(* CODESYS project PLC_241_14_11_2020.project
   Title: PLC_241
   Version: 0.0.0.0
   Author: anvar

Project tree, tasks and I/O mapping:
  PLC_241 : TM241CE40T/U, Schneider Electric, order no. TM241CE40T/U, version 4.0.6.18
    application Application
      task MAST (cyclic, interval 20 ms, priority 15, watchdog 100 ms x 1) calls BIND, prgLoad, prgLoad_K, prgAdd_weight, CONVERT_REAL_TO_INT, prgDOSING_BIG_WEIGHT, Recept, MotoHours, vsState
      global variables GVL
      global variables IN_OUT
      global variables Mechanizm
      program BIND [ST]
      data type Real_word
      FB/
        SH/
          function block Z [LD]
        Flap/
          function block KP [LD]
        Noria/
          function block N [LD]
        SKTR/
          function block T [LD]
          function block Shnek [LD]
          function block Dozator [LD]
        ASP/
          function block AC [LD]
          function block shluz [LD]
        vibr/
          function block VB [LD]
        scalperator/
          function block SCLP [LD]
      POU/
        program prgLoad [LD]
        program prgLoad_K [LD]
        program prgAdd_weight [LD]
        program prgDOSING_BIG_WEIGHT [LD]
        program MotoHours [ST]
      global variables ErrList
      global variables Pozition_flap
      program Recept [ST]
      program CONVERT_REAL_TO_INT [ST]
      global variables PersistentVars
      program vsState [ST]
      function funStepMH [ST]
    DI : Digital Inputs, Schneider Electric, version 4.0.6.18
        input  idwDI_IDW0 : DWORD  // IDW0
        input  Application.x0_0 : BOOL  // IDW0.I0
        input  Application.x0_1 : BOOL  // IDW0.I1
        input  Application.x0_2 : BOOL  // IDW0.I2
        input  Application.x0_3 : BOOL  // IDW0.I3
        input  Application.x0_4 : BOOL  // IDW0.I4
        input  Application.x0_5 : BOOL  // IDW0.I5
        input  Application.x0_6 : BOOL  // IDW0.I6
        input  Application.x0_7 : BOOL  // IDW0.I7
        input  Application.x0_8 : BOOL  // IDW0.I8
        input  Application.x0_9 : BOOL  // IDW0.I9
        input  Application.x0_10 : BOOL  // IDW0.I10
        input  Application.x0_11 : BOOL  // IDW0.I11
        input  Application.x0_12 : BOOL  // IDW0.I12
        input  Application.x0_13 : BOOL  // IDW0.I13
        input  Application.x0_14 : BOOL  // IDW0.I14
        input  Application.x0_15 : BOOL  // IDW0.I15
        input  Application.x0_16 : BOOL  // IDW0.I16
        input  Application.x0_17 : BOOL  // IDW0.I17
        input  Application.x0_18 : BOOL  // IDW0.I18
        input  Application.x0_19 : BOOL  // IDW0.I19
        input  Application.x0_20 : BOOL  // IDW0.I20
        input  Application.x0_21 : BOOL  // IDW0.I21
        input  Application.x0_22 : BOOL  // IDW0.I22
        input  Application.x0_23 : BOOL  // IDW0.I23
        input  ibDI_IB1 : BYTE  // IB1
    DQ : Digital Outputs, Schneider Electric, version 4.0.6.18
        output Application.y0_0 : BOOL  // QW0.Q0
        output Application.y0_1 : BOOL  // QW0.Q1
        output Application.y0_2 : BOOL  // QW0.Q2
        output Application.y0_3 : BOOL  // QW0.Q3
        output Application.y0_4 : BOOL  // QW0.Q4
        output Application.y0_5 : BOOL  // QW0.Q5
        output Application.y0_6 : BOOL  // QW0.Q6
        output Application.y0_7 : BOOL  // QW0.Q7
        output Application.y0_8 : BOOL  // QW0.Q8
        output Application.y0_9 : BOOL  // QW0.Q9
        output Application.y0_10 : BOOL  // QW0.Q10
        output Application.y0_11 : BOOL  // QW0.Q11
        output Application.y0_12 : BOOL  // QW0.Q12
        output Application.y0_13 : BOOL  // QW0.Q13
        output Application.y0_14 : BOOL  // QW0.Q14
        output Application.y0_15 : BOOL  // QW0.Q15
        output qbDQ_QB1 : BYTE  // QB1
        unmapped channels: QW0
    Counters : Counters, Schneider Electric, version 4.0.6.18
    Pulse_Generators : Pulse Generators, Schneider Electric, version 4.0.6.18
    Cartridge_1 : Cartridge, Schneider Electric, version 4.0.6.18
    Cartridge_2 : Cartridge, Schneider Electric, version 4.0.6.18
    IO_Bus : IO bus - TM3, Schneider Electric, version 4.0.6.18
      IN_1 : TM3DI32K, Schneider Electric, order no. TM3DI32K, version 1.0.1.3
          input  idwIN_1_ID0 : DWORD  // ID0
          input  Application.x1_0 : BOOL  // ID0.I0
          input  Application.x1_1 : BOOL  // ID0.I1
          input  Application.x1_2 : BOOL  // ID0.I2
          input  Application.x1_3 : BOOL  // ID0.I3
          input  Application.x1_4 : BOOL  // ID0.I4
          input  Application.x1_5 : BOOL  // ID0.I5
          input  Application.x1_6 : BOOL  // ID0.I6
          input  Application.x1_7 : BOOL  // ID0.I7
          input  Application.x1_8 : BOOL  // ID0.I8
          input  Application.x1_9 : BOOL  // ID0.I9
          input  Application.x1_10 : BOOL  // ID0.I10
          input  Application.x1_11 : BOOL  // ID0.I11
          input  Application.x1_12 : BOOL  // ID0.I12
          input  Application.x1_13 : BOOL  // ID0.I13
          input  Application.x1_14 : BOOL  // ID0.I14
          input  Application.x1_15 : BOOL  // ID0.I15
          input  Application.x1_16 : BOOL  // ID0.I16
          input  Application.x1_17 : BOOL  // ID0.I17
          input  Application.x1_18 : BOOL  // ID0.I18
          input  Application.x1_19 : BOOL  // ID0.I19
          input  Application.x1_20 : BOOL  // ID0.I20
          input  Application.x1_21 : BOOL  // ID0.I21
          input  Application.x1_22 : BOOL  // ID0.I22
          input  Application.x1_23 : BOOL  // ID0.I23
          input  Application.x1_24 : BOOL  // ID0.I24
          input  Application.x1_25 : BOOL  // ID0.I25
          input  Application.x1_26 : BOOL  // ID0.I26
          input  Application.x1_27 : BOOL  // ID0.I27
          input  Application.x1_28 : BOOL  // ID0.I28
          input  Application.x1_29 : BOOL  // ID0.I29
          input  Application.x1_30 : BOOL  // ID0.I30
          input  Application.x1_31 : BOOL  // ID0.I31
      IN_2 : TM3DI32K, Schneider Electric, order no. TM3DI32K, version 1.0.1.3
          input  idwIN_2_ID0 : DWORD  // ID0
          input  Application.x2_0 : BOOL  // ID0.I0
          input  Application.x2_1 : BOOL  // ID0.I1
          input  Application.x2_2 : BOOL  // ID0.I2
          input  Application.x2_3 : BOOL  // ID0.I3
          input  Application.x2_4 : BOOL  // ID0.I4
          input  Application.x2_5 : BOOL  // ID0.I5
          input  Application.x2_6 : BOOL  // ID0.I6
          input  Application.x2_7 : BOOL  // ID0.I7
          input  Application.x2_8 : BOOL  // ID0.I8
          input  Application.x2_9 : BOOL  // ID0.I9
          input  Application.x2_10 : BOOL  // ID0.I10
          input  Application.x2_11 : BOOL  // ID0.I11
          input  Application.x2_12 : BOOL  // ID0.I12
          input  Application.x2_13 : BOOL  // ID0.I13
          input  Application.x2_14 : BOOL  // ID0.I14
          input  Application.x2_15 : BOOL  // ID0.I15
          input  Application.x2_16 : BOOL  // ID0.I16
          input  Application.x2_17 : BOOL  // ID0.I17
          input  Application.x2_18 : BOOL  // ID0.I18
          input  Application.x2_19 : BOOL  // ID0.I19
          input  Application.x2_20 : BOOL  // ID0.I20
          input  Application.x2_21 : BOOL  // ID0.I21
          input  Application.x2_22 : BOOL  // ID0.I22
          input  Application.x2_23 : BOOL  // ID0.I23
          input  Application.x2_24 : BOOL  // ID0.I24
          input  Application.x2_25 : BOOL  // ID0.I25
          input  Application.x2_26 : BOOL  // ID0.I26
          input  Application.x2_27 : BOOL  // ID0.I27
          input  Application.x2_28 : BOOL  // ID0.I28
          input  Application.x2_29 : BOOL  // ID0.I29
          input  Application.x2_30 : BOOL  // ID0.I30
          input  Application.x2_31 : BOOL  // ID0.I31
      IN_3 : TM3DI32K, Schneider Electric, order no. TM3DI32K, version 1.0.1.3
          input  idwIN_3_ID0 : DWORD  // ID0
          input  Application.x3_0 : BOOL  // ID0.I0
          input  Application.x3_1 : BOOL  // ID0.I1
          input  Application.x3_2 : BOOL  // ID0.I2
          input  Application.x3_3 : BOOL  // ID0.I3
          input  Application.x3_4 : BOOL  // ID0.I4
          input  Application.x3_5 : BOOL  // ID0.I5
          input  Application.x3_6 : BOOL  // ID0.I6
          input  Application.x3_7 : BOOL  // ID0.I7
          input  Application.x3_8 : BOOL  // ID0.I8
          input  Application.x3_9 : BOOL  // ID0.I9
          input  Application.x3_10 : BOOL  // ID0.I10
          input  Application.x3_11 : BOOL  // ID0.I11
          input  Application.x3_12 : BOOL  // ID0.I12
          input  Application.x3_13 : BOOL  // ID0.I13
          input  Application.x3_14 : BOOL  // ID0.I14
          input  Application.x3_15 : BOOL  // ID0.I15
          input  Application.x3_16 : BOOL  // ID0.I16
          input  Application.x3_17 : BOOL  // ID0.I17
          input  Application.x3_18 : BOOL  // ID0.I18
          input  Application.x3_19 : BOOL  // ID0.I19
          input  Application.x3_20 : BOOL  // ID0.I20
          input  Application.x3_21 : BOOL  // ID0.I21
          input  Application.x3_22 : BOOL  // ID0.I22
          input  Application.x3_23 : BOOL  // ID0.I23
          input  Application.x3_24 : BOOL  // ID0.I24
          input  Application.x3_25 : BOOL  // ID0.I25
          input  Application.x3_26 : BOOL  // ID0.I26
          input  Application.x3_27 : BOOL  // ID0.I27
          input  Application.x3_28 : BOOL  // ID0.I28
          input  Application.x3_29 : BOOL  // ID0.I29
          input  Application.x3_30 : BOOL  // ID0.I30
          input  Application.x3_31 : BOOL  // ID0.I31
      IN_4 : TM3DI32K, Schneider Electric, order no. TM3DI32K, version 1.0.1.3
          input  idwIN_4_ID0 : DWORD  // ID0
          input  Application.x4_0 : BOOL  // ID0.I0
          input  Application.x4_1 : BOOL  // ID0.I1
          input  Application.x4_2 : BOOL  // ID0.I2
          input  Application.x4_3 : BOOL  // ID0.I3
          input  Application.x4_4 : BOOL  // ID0.I4
          input  Application.x4_5 : BOOL  // ID0.I5
          input  Application.x4_6 : BOOL  // ID0.I6
          input  Application.x4_7 : BOOL  // ID0.I7
          input  Application.x4_8 : BOOL  // ID0.I8
          input  Application.x4_9 : BOOL  // ID0.I9
          input  Application.x4_10 : BOOL  // ID0.I10
          input  Application.x4_11 : BOOL  // ID0.I11
          input  Application.x4_12 : BOOL  // ID0.I12
          input  Application.x4_13 : BOOL  // ID0.I13
          input  Application.x4_14 : BOOL  // ID0.I14
          input  Application.x4_15 : BOOL  // ID0.I15
          input  Application.x4_16 : BOOL  // ID0.I16
          input  Application.x4_17 : BOOL  // ID0.I17
          input  Application.x4_18 : BOOL  // ID0.I18
          input  Application.x4_19 : BOOL  // ID0.I19
          input  Application.x4_20 : BOOL  // ID0.I20
          input  Application.x4_21 : BOOL  // ID0.I21
          input  Application.x4_22 : BOOL  // ID0.I22
          input  Application.x4_23 : BOOL  // ID0.I23
          input  Application.x4_24 : BOOL  // ID0.I24
          input  Application.x4_25 : BOOL  // ID0.I25
          input  Application.x4_26 : BOOL  // ID0.I26
          input  Application.x4_27 : BOOL  // ID0.I27
          input  Application.x4_28 : BOOL  // ID0.I28
          input  Application.x4_29 : BOOL  // ID0.I29
          input  Application.x4_30 : BOOL  // ID0.I30
          input  Application.x4_31 : BOOL  // ID0.I31
      IN_5 : TM3DI32K, Schneider Electric, order no. TM3DI32K, version 1.0.1.3
          input  idwIN_5_ID0 : DWORD  // ID0
          input  Application.x5_0 : BOOL  // ID0.I0
          input  Application.x5_1 : BOOL  // ID0.I1
          input  Application.x5_2 : BOOL  // ID0.I2
          input  Application.x5_3 : BOOL  // ID0.I3
          input  Application.x5_4 : BOOL  // ID0.I4
          input  Application.x5_5 : BOOL  // ID0.I5
          input  Application.x5_6 : BOOL  // ID0.I6
          input  Application.x5_7 : BOOL  // ID0.I7
          input  Application.x5_8 : BOOL  // ID0.I8
          input  Application.x5_9 : BOOL  // ID0.I9
          input  Application.x5_10 : BOOL  // ID0.I10
          input  Application.x5_11 : BOOL  // ID0.I11
          input  Application.x5_12 : BOOL  // ID0.I12
          input  Application.x5_13 : BOOL  // ID0.I13
          input  Application.x5_14 : BOOL  // ID0.I14
          input  Application.x5_15 : BOOL  // ID0.I15
          input  Application.x5_16 : BOOL  // ID0.I16
          input  Application.x5_17 : BOOL  // ID0.I17
          input  Application.x5_18 : BOOL  // ID0.I18
          input  Application.x5_19 : BOOL  // ID0.I19
          input  Application.x5_20 : BOOL  // ID0.I20
          input  Application.x5_21 : BOOL  // ID0.I21
          input  Application.x5_22 : BOOL  // ID0.I22
          input  Application.x5_23 : BOOL  // ID0.I23
          input  Application.x5_24 : BOOL  // ID0.I24
          input  Application.x5_25 : BOOL  // ID0.I25
          input  Application.x5_26 : BOOL  // ID0.I26
          input  Application.x5_27 : BOOL  // ID0.I27
          input  Application.x5_28 : BOOL  // ID0.I28
          input  Application.x5_29 : BOOL  // ID0.I29
          input  Application.x5_30 : BOOL  // ID0.I30
          input  Application.x5_31 : BOOL  // ID0.I31
      OUT_6 : TM3DQ32TK, Schneider Electric, order no. TM3DQ32TK, version 1.0.1.3
          output Application.y6_0 : BOOL  // QD0.Q0
          output Application.y6_1 : BOOL  // QD0.Q1
          output Application.y6_2 : BOOL  // QD0.Q2
          output Application.y6_3 : BOOL  // QD0.Q3
          output Application.y6_4 : BOOL  // QD0.Q4
          output Application.y6_5 : BOOL  // QD0.Q5
          output Application.y6_6 : BOOL  // QD0.Q6
          output Application.y6_7 : BOOL  // QD0.Q7
          output Application.y6_8 : BOOL  // QD0.Q8
          output Application.y6_9 : BOOL  // QD0.Q9
          output Application.y6_10 : BOOL  // QD0.Q10
          output Application.y6_11 : BOOL  // QD0.Q11
          output Application.y6_12 : BOOL  // QD0.Q12
          output Application.y6_13 : BOOL  // QD0.Q13
          output Application.y6_14 : BOOL  // QD0.Q14
          output Application.y6_15 : BOOL  // QD0.Q15
          output Application.y6_16 : BOOL  // QD0.Q16
          output Application.y6_17 : BOOL  // QD0.Q17
          output Application.y6_18 : BOOL  // QD0.Q18
          output Application.y6_19 : BOOL  // QD0.Q19
          output Application.y6_20 : BOOL  // QD0.Q20
          output Application.y6_21 : BOOL  // QD0.Q21
          output Application.y6_22 : BOOL  // QD0.Q22
          output Application.y6_23 : BOOL  // QD0.Q23
          output Application.y6_24 : BOOL  // QD0.Q24
          output Application.y6_25 : BOOL  // QD0.Q25
          output Application.y6_26 : BOOL  // QD0.Q26
          output Application.y6_27 : BOOL  // QD0.Q27
          output Application.y6_28 : BOOL  // QD0.Q28
          output Application.y6_29 : BOOL  // QD0.Q29
          output Application.y6_30 : BOOL  // QD0.Q30
          output Application.y6_31 : BOOL  // QD0.Q31
          unmapped channels: QD0
      OUT_7 : TM3DQ32TK, Schneider Electric, order no. TM3DQ32TK, version 1.0.1.3
          output Application.y7_0 : BOOL  // QD0.Q0
          output Application.y7_1 : BOOL  // QD0.Q1
          output Application.y7_2 : BOOL  // QD0.Q2
          output Application.y7_3 : BOOL  // QD0.Q3
          output Application.y7_4 : BOOL  // QD0.Q4
          output Application.y7_5 : BOOL  // QD0.Q5
          output Application.y7_6 : BOOL  // QD0.Q6
          output Application.y7_7 : BOOL  // QD0.Q7
          output Application.y7_8 : BOOL  // QD0.Q8
          output Application.y7_9 : BOOL  // QD0.Q9
          output Application.y7_10 : BOOL  // QD0.Q10
          output Application.y7_11 : BOOL  // QD0.Q11
          output Application.y7_12 : BOOL  // QD0.Q12
          output Application.y7_13 : BOOL  // QD0.Q13
          output Application.y7_14 : BOOL  // QD0.Q14
          output Application.y7_15 : BOOL  // QD0.Q15
          output Application.y7_16 : BOOL  // QD0.Q16
          output Application.y7_17 : BOOL  // QD0.Q17
          output Application.y7_18 : BOOL  // QD0.Q18
          output Application.y7_19 : BOOL  // QD0.Q19
          output Application.y7_20 : BOOL  // QD0.Q20
          output Application.y7_21 : BOOL  // QD0.Q21
          output Application.y7_22 : BOOL  // QD0.Q22
          output Application.y7_23 : BOOL  // QD0.Q23
          output Application.y7_24 : BOOL  // QD0.Q24
          output Application.y7_25 : BOOL  // QD0.Q25
          output Application.y7_26 : BOOL  // QD0.Q26
          output Application.y7_27 : BOOL  // QD0.Q27
          output Application.y7_28 : BOOL  // QD0.Q28
          output Application.y7_29 : BOOL  // QD0.Q29
          output Application.y7_30 : BOOL  // QD0.Q30
          output Application.y7_31 : BOOL  // QD0.Q31
          unmapped channels: QD0
    COM_Bus : COM bus, Schneider Electric, version 4.0.6.18
    Ethernet_1 : Ethernet Network, Schneider Electric, version 4.0.6.18
        settings: IPAddress = [192, 168, 3, 241]; SubnetMask = [255, 255, 255, 0]; WebServer = TRUE; FTP Server = TRUE; SoMachine Protocol = TRUE; Modbus Server = TRUE; NetManage Protocol = TRUE; SNMP protocol = TRUE; Enable Routing = FALSE; WebVisu protocol = TRUE; DHCP Server Active = TRUE
      Ethernet_Manager : Industrial Ethernet Manager, Schneider Electric, version 1.0.12.21
          settings: BinaryFileSize = 396; Dhcps Host 0.Client Mac Address = [16#0, 16#0, 16#0, 16#0, 16#0]; Dhcps Host 0.Client Device Name = 'DEVICE_1'; Dhcps Host 0.Client IP Address = [192, 168, 3, 221]; Dhcps Host 0.Network Mask = [255, 255, 255, 0]; Dhcps Host 0.Default Gateway = [192, 168, 3, 241]; Dhcps Host 1.Client Mac Address = [16#0, 16#0, 16#0, 16#0, 16#0]; Dhcps Host 2.Client Mac Address = [16#0, 16#0, 16#0, 16#0, 16#0]; Dhcps Host 3.Client Mac Address = [16#0, 16#0, 16#0, 16#0, 16#0]; Dhcps Host 4.Client Mac Address = [16#0, 16#0, 16#0, 16#0, 16#0]; Dhcps Host 5.Client Mac Address = [16#0, 16#0, 16#0, 16#0, 16#0]; Dhcps Host 6.Client Mac Address = [16#0, 16#0, 16#0, 16#0, 16#0]; Dhcps Host 7.Client Mac Address = [16#0, 16#0, 16#0, 16#0, 16#0]; Dhcps Host 8.Client Mac Address = [16#0, 16#0, 16#0, 16#0, 16#0]; Dhcps Host 9.Client Mac Address = [16#0, 16#0, 16#0, 16#0, 16#0]; Dhcps Host 10.Client Mac Address = [16#0, 16#0, 16#0, 16#0, 16#0]; Dhcps Host 11.Client Mac Address = [16#0, 16#0, 16#0, 16#0, 16#0]; Dhcps Host 12.Client Mac Address = [16#0, 16#0, 16#0, 16#0, 16#0]; Dhcps Host 13.Client Mac Address = [16#0, 16#0, 16#0, 16#0, 16#0]; Dhcps Host 14.Client Mac Address = [16#0, 16#0, 16#0, 16#0, 16#0]; Dhcps Host 15.Client Mac Address = [16#0, 16#0, 16#0, 16#0, 16#0]; Dhcps Host 16.Client Mac Address = [16#0, 16#0, 16#0, 16#0, 16#0]; Dhcps Host 17.Client Mac Address = [16#0, 16#0, 16#0, 16#0, 16#0]; Dhcps Host 18.Client Mac Address = [16#0, 16#0, 16#0, 16#0, 16#0]; Dhcps Host 19.Client Mac Address = [16#0, 16#0, 16#0, 16#0, 16#0]; Dhcps Host 20.Client Mac Address = [16#0, 16#0, 16#0, 16#0, 16#0]; Dhcps Host 21.Client Mac Address = [16#0, 16#0, 16#0, 16#0, 16#0]; Dhcps Host 22.Client Mac Address = [16#0, 16#0, 16#0, 16#0, 16#0]; Dhcps Host 23.Client Mac Address = [16#0, 16#0, 16#0, 16#0, 16#0]; Dhcps Host 24.Client Mac Address = [16#0, 16#0, 16#0, 16#0, 16#0]; Dhcps Host 25.Client Mac Address = [16#0, 16#0, 16#0, 16#0, 16#0]; Dhcps Host 26.Client Mac Address = [16#0, 16#0, 16#0, 16#0, 16#0]; Dhcps Host 27.Client Mac Address = [16#0, 16#0, 16#0, 16#0, 16#0]; Dhcps Host 28.Client Mac Address = [16#0, 16#0, 16#0, 16#0, 16#0]; Dhcps Host 29.Client Mac Address = [16#0, 16#0, 16#0, 16#0, 16#0]; Dhcps Host 30.Client Mac Address = [16#0, 16#0, 16#0, 16#0, 16#0]; Dhcps Host 31.Client Mac Address = [16#0, 16#0, 16#0, 16#0, 16#0]; Dhcps Host 32.Client Mac Address = [16#0, 16#0, 16#0, 16#0, 16#0]; Dhcps Host 33.Client Mac Address = [16#0, 16#0, 16#0, 16#0, 16#0]; Dhcps Host 34.Client Mac Address = [16#0, 16#0, 16#0, 16#0, 16#0];
            Dhcps Host 35.Client Mac Address = [16#0, 16#0, 16#0, 16#0, 16#0]; Dhcps Host 36.Client Mac Address = [16#0, 16#0, 16#0, 16#0, 16#0]; Dhcps Host 37.Client Mac Address = [16#0, 16#0, 16#0, 16#0, 16#0]; Dhcps Host 38.Client Mac Address = [16#0, 16#0, 16#0, 16#0, 16#0]; Dhcps Host 39.Client Mac Address = [16#0, 16#0, 16#0, 16#0, 16#0]; Dhcps Host 40.Client Mac Address = [16#0, 16#0, 16#0, 16#0, 16#0]; Dhcps Host 41.Client Mac Address = [16#0, 16#0, 16#0, 16#0, 16#0]; Dhcps Host 42.Client Mac Address = [16#0, 16#0, 16#0, 16#0, 16#0]; Dhcps Host 43.Client Mac Address = [16#0, 16#0, 16#0, 16#0, 16#0]; Dhcps Host 44.Client Mac Address = [16#0, 16#0, 16#0, 16#0, 16#0]; Dhcps Host 45.Client Mac Address = [16#0, 16#0, 16#0, 16#0, 16#0]; Dhcps Host 46.Client Mac Address = [16#0, 16#0, 16#0, 16#0, 16#0]; Dhcps Host 47.Client Mac Address = [16#0, 16#0, 16#0, 16#0, 16#0]; Dhcps Host 48.Client Mac Address = [16#0, 16#0, 16#0, 16#0, 16#0]; Dhcps Host 49.Client Mac Address = [16#0, 16#0, 16#0, 16#0, 16#0]; Dhcps Host 50.Client Mac Address = [16#0, 16#0, 16#0, 16#0, 16#0]; Dhcps Host 51.Client Mac Address = [16#0, 16#0, 16#0, 16#0, 16#0]; Dhcps Host 52.Client Mac Address = [16#0, 16#0, 16#0, 16#0, 16#0]; Dhcps Host 53.Client Mac Address = [16#0, 16#0, 16#0, 16#0, 16#0]; Dhcps Host 54.Client Mac Address = [16#0, 16#0, 16#0, 16#0, 16#0]; Dhcps Host 55.Client Mac Address = [16#0, 16#0, 16#0, 16#0, 16#0]; Dhcps Host 56.Client Mac Address = [16#0, 16#0, 16#0, 16#0, 16#0]; Dhcps Host 57.Client Mac Address = [16#0, 16#0, 16#0, 16#0, 16#0]; Dhcps Host 58.Client Mac Address = [16#0, 16#0, 16#0, 16#0, 16#0]; Dhcps Host 59.Client Mac Address = [16#0, 16#0, 16#0, 16#0, 16#0]; Dhcps Host 60.Client Mac Address = [16#0, 16#0, 16#0, 16#0, 16#0]; Dhcps Host 61.Client Mac Address = [16#0, 16#0, 16#0, 16#0, 16#0]; Dhcps Host 62.Client Mac Address = [16#0, 16#0, 16#0, 16#0, 16#0]; Dhcps Host 63.Client Mac Address = [16#0, 16#0, 16#0, 16#0, 16#0]; Dhcps Host 64.Client Mac Address = [16#0, 16#0, 16#0, 16#0, 16#0]; Dhcps Host 65.Client Mac Address = [16#0, 16#0, 16#0, 16#0, 16#0]; Dhcps Host 66.Client Mac Address = [16#0, 16#0, 16#0, 16#0, 16#0]; Dhcps Host 67.Client Mac Address = [16#0, 16#0, 16#0, 16#0, 16#0]; Dhcps Host 68.Client Mac Address = [16#0, 16#0, 16#0, 16#0, 16#0]; Dhcps Host 69.Client Mac Address = [16#0, 16#0, 16#0, 16#0, 16#0]; Dhcps Host 70.Client Mac Address = [16#0, 16#0, 16#0, 16#0, 16#0]; Dhcps Host 71.Client Mac Address = [16#0, 16#0, 16#0, 16#0, 16#0]; Dhcps Host 72.Client Mac Address = [16#0, 16#0, 16#0, 16#0, 16#0]; Dhcps Host 73.Client Mac Address = [16#0, 16#0, 16#0, 16#0, 16#0]; Dhcps Host 74.Client Mac Address = [16#0, 16#0, 16#0, 16#0, 16#0];
            Dhcps Host 75.Client Mac Address = [16#0, 16#0, 16#0, 16#0, 16#0]; Dhcps Host 76.Client Mac Address = [16#0, 16#0, 16#0, 16#0, 16#0]; Dhcps Host 77.Client Mac Address = [16#0, 16#0, 16#0, 16#0, 16#0]; Dhcps Host 78.Client Mac Address = [16#0, 16#0, 16#0, 16#0, 16#0]; Dhcps Host 79.Client Mac Address = [16#0, 16#0, 16#0, 16#0, 16#0]; Dhcps Host 80.Client Mac Address = [16#0, 16#0, 16#0, 16#0, 16#0]; Dhcps Host 81.Client Mac Address = [16#0, 16#0, 16#0, 16#0, 16#0]; Dhcps Host 82.Client Mac Address = [16#0, 16#0, 16#0, 16#0, 16#0]; Dhcps Host 83.Client Mac Address = [16#0, 16#0, 16#0, 16#0, 16#0]; Dhcps Host 84.Client Mac Address = [16#0, 16#0, 16#0, 16#0, 16#0]; Dhcps Host 85.Client Mac Address = [16#0, 16#0, 16#0, 16#0, 16#0]; Dhcps Host 86.Client Mac Address = [16#0, 16#0, 16#0, 16#0, 16#0]; Dhcps Host 87.Client Mac Address = [16#0, 16#0, 16#0, 16#0, 16#0]; Dhcps Host 88.Client Mac Address = [16#0, 16#0, 16#0, 16#0, 16#0]; Dhcps Host 89.Client Mac Address = [16#0, 16#0, 16#0, 16#0, 16#0]; Dhcps Host 90.Client Mac Address = [16#0, 16#0, 16#0, 16#0, 16#0]; Dhcps Host 91.Client Mac Address = [16#0, 16#0, 16#0, 16#0, 16#0]; Dhcps Host 92.Client Mac Address = [16#0, 16#0, 16#0, 16#0, 16#0]; Dhcps Host 93.Client Mac Address = [16#0, 16#0, 16#0, 16#0, 16#0]; Dhcps Host 94.Client Mac Address = [16#0, 16#0, 16#0, 16#0, 16#0]; Dhcps Host 95.Client Mac Address = [16#0, 16#0, 16#0, 16#0, 16#0]; Dhcps Host 96.Client Mac Address = [16#0, 16#0, 16#0, 16#0, 16#0]; Dhcps Host 97.Client Mac Address = [16#0, 16#0, 16#0, 16#0, 16#0]; Dhcps Host 98.Client Mac Address = [16#0, 16#0, 16#0, 16#0, 16#0]; Dhcps Host 99.Client Mac Address = [16#0, 16#0, 16#0, 16#0, 16#0]; Dhcps Host 100.Client Mac Address = [16#0, 16#0, 16#0, 16#0, 16#0]; Dhcps Host 101.Client Mac Address = [16#0, 16#0, 16#0, 16#0, 16#0]; Dhcps Host 102.Client Mac Address = [16#0, 16#0, 16#0, 16#0, 16#0]; Dhcps Host 103.Client Mac Address = [16#0, 16#0, 16#0, 16#0, 16#0]; Dhcps Host 104.Client Mac Address = [16#0, 16#0, 16#0, 16#0, 16#0]; Dhcps Host 105.Client Mac Address = [16#0, 16#0, 16#0, 16#0, 16#0]; Dhcps Host 106.Client Mac Address = [16#0, 16#0, 16#0, 16#0, 16#0]; Dhcps Host 107.Client Mac Address = [16#0, 16#0, 16#0, 16#0, 16#0]; Dhcps Host 108.Client Mac Address = [16#0, 16#0, 16#0, 16#0, 16#0]; Dhcps Host 109.Client Mac Address = [16#0, 16#0, 16#0, 16#0, 16#0]; Dhcps Host 110.Client Mac Address = [16#0, 16#0, 16#0, 16#0, 16#0]; Dhcps Host 111.Client Mac Address = [16#0, 16#0, 16#0, 16#0, 16#0]; Dhcps Host 112.Client Mac Address = [16#0, 16#0, 16#0, 16#0, 16#0]; Dhcps Host 113.Client Mac Address = [16#0, 16#0, 16#0, 16#0, 16#0]; Dhcps Host 114.Client Mac Address = [16#0, 16#0, 16#0, 16#0, 16#0];
            Dhcps Host 115.Client Mac Address = [16#0, 16#0, 16#0, 16#0, 16#0]; Dhcps Host 116.Client Mac Address = [16#0, 16#0, 16#0, 16#0, 16#0]; Dhcps Host 117.Client Mac Address = [16#0, 16#0, 16#0, 16#0, 16#0]; Dhcps Host 118.Client Mac Address = [16#0, 16#0, 16#0, 16#0, 16#0]; Dhcps Host 119.Client Mac Address = [16#0, 16#0, 16#0, 16#0, 16#0]; Dhcps Host 120.Client Mac Address = [16#0, 16#0, 16#0, 16#0, 16#0]; Dhcps Host 121.Client Mac Address = [16#0, 16#0, 16#0, 16#0, 16#0]; Dhcps Host 122.Client Mac Address = [16#0, 16#0, 16#0, 16#0, 16#0]; Dhcps Host 123.Client Mac Address = [16#0, 16#0, 16#0, 16#0, 16#0]; Dhcps Host 124.Client Mac Address = [16#0, 16#0, 16#0, 16#0, 16#0]; Dhcps Host 125.Client Mac Address = [16#0, 16#0, 16#0, 16#0, 16#0]; Dhcps Host 126.Client Mac Address = [16#0, 16#0, 16#0, 16#0, 16#0]; Dhcps Host 127.Client Mac Address = [16#0, 16#0, 16#0, 16#0, 16#0]; Dhcps Host 128.Client Mac Address = [16#0, 16#0, 16#0, 16#0, 16#0]; serialized Values = 9e259374-7d59-4259-90d2-1eb457ee1159=0|
          unmapped channels: Global Status, Healthbit 0, Healthbit 1, Healthbit 2, Healthbit 3
        Modbus_TCP_Slave_PLC221 : Generic Modbus TCP Slave, Schneider Electric, version 1.0.2.21
            settings: Unit-ID = 248; IPAddress = [192, 168, 3, 221]; GatewayAddress = [192, 168, 3, 241]; DeviceName = 'DEVICE_1'; PLC221.Channel ID = 0; PLC221.Unit-ID = 255; PLC221.Repetition Rate = 20; PLC221.Function Code = 23; PLC221.Read Offset = 16#0000; PLC221.Read Length = 20; PLC221.Write Offset = 16#0014; PLC221.Write Length = 10
            input  Application.a2x0_0 : BOOL  // PLC221.Bit 0
            input  Application.a2x0_1 : BOOL  // PLC221.Bit 1
            input  Application.a2x0_2 : BOOL  // PLC221.Bit 2
            input  Application.a2x0_3 : BOOL  // PLC221.Bit 3
            input  Application.a2x0_4 : BOOL  // PLC221.Bit 4
            input  Application.a2x0_5 : BOOL  // PLC221.Bit 5
            input  Application.a2x0_6 : BOOL  // PLC221.Bit 6
            input  Application.a2x0_7 : BOOL  // PLC221.Bit 7
            input  Application.a2x0_8 : BOOL  // PLC221.Bit 8
            input  Application.a2x0_9 : BOOL  // PLC221.Bit 9
            input  Application.a2x0_10 : BOOL  // PLC221.Bit 10
            input  Application.a2x0_11 : BOOL  // PLC221.Bit 11
            input  Application.a2x0_12 : BOOL  // PLC221.Bit 12
            input  Application.a2x0_13 : BOOL  // PLC221.Bit 13
            input  Application.a2x0_14 : BOOL  // PLC221.Bit 14
            input  Application.a2x0_15 : BOOL  // PLC221.Bit 15
            input  Application.a2x0_16 : BOOL  // PLC221.Bit 0
            input  Application.a2x0_17 : BOOL  // PLC221.Bit 1
            input  Application.a2x0_18 : BOOL  // PLC221.Bit 2
            input  Application.a2x0_19 : BOOL  // PLC221.Bit 3
            input  Application.a2x0_20 : BOOL  // PLC221.Bit 4
            input  Application.a2x0_21 : BOOL  // PLC221.Bit 5
            input  Application.a2x0_22 : BOOL  // PLC221.Bit 6
            input  Application.a2x0_23 : BOOL  // PLC221.Bit 7
            input  Application.a2x3_0 : BOOL  // PLC221.Bit 0
            input  Application.a2x3_1 : BOOL  // PLC221.Bit 1
            input  Application.a2x3_2 : BOOL  // PLC221.Bit 2
            input  Application.a2x3_3 : BOOL  // PLC221.Bit 3
            input  Application.a2x3_4 : BOOL  // PLC221.Bit 4
            input  Application.a2x3_5 : BOOL  // PLC221.Bit 5
            input  Application.a2x3_6 : BOOL  // PLC221.Bit 6
            input  Application.a2x3_7 : BOOL  // PLC221.Bit 7
            input  Application.a2x3_8 : BOOL  // PLC221.Bit 8
            input  Application.a2x3_9 : BOOL  // PLC221.Bit 9
            input  Application.a2x3_10 : BOOL  // PLC221.Bit 10
            input  Application.a2x3_11 : BOOL  // PLC221.Bit 11
            input  Application.a2x3_12 : BOOL  // PLC221.Bit 12
            input  Application.a2x3_13 : BOOL  // PLC221.Bit 13
            input  Application.a2x3_14 : BOOL  // PLC221.Bit 14
            input  Application.a2x3_15 : BOOL  // PLC221.Bit 15
            input  Application.a2x3_16 : BOOL  // PLC221.Bit 0
            input  Application.a2x3_17 : BOOL  // PLC221.Bit 1
            input  Application.a2x3_18 : BOOL  // PLC221.Bit 2
            input  Application.a2x3_19 : BOOL  // PLC221.Bit 3
            input  Application.a2x3_20 : BOOL  // PLC221.Bit 4
            input  Application.a2x3_21 : BOOL  // PLC221.Bit 5
            input  Application.a2x3_22 : BOOL  // PLC221.Bit 6
            input  Application.a2x3_23 : BOOL  // PLC221.Bit 7
            input  Application.a2x3_24 : BOOL  // PLC221.Bit 8
            input  Application.a2x3_25 : BOOL  // PLC221.Bit 9
            input  Application.a2x3_26 : BOOL  // PLC221.Bit 10
            input  Application.a2x3_27 : BOOL  // PLC221.Bit 11
            input  Application.a2x3_28 : BOOL  // PLC221.Bit 12
            input  Application.a2x3_29 : BOOL  // PLC221.Bit 13
            input  Application.a2x3_30 : BOOL  // PLC221.Bit 14
            input  Application.a2x3_31 : BOOL  // PLC221.Bit 15
            input  Application.a2x4_0 : BOOL  // PLC221.Bit 0
            input  Application.a2x4_1 : BOOL  // PLC221.Bit 1
            input  Application.a2x4_2 : BOOL  // PLC221.Bit 2
            input  Application.a2x4_3 : BOOL  // PLC221.Bit 3
            input  Application.a2x4_4 : BOOL  // PLC221.Bit 4
            input  Application.a2x4_5 : BOOL  // PLC221.Bit 5
            input  Application.a2x4_6 : BOOL  // PLC221.Bit 6
            input  Application.a2x4_7 : BOOL  // PLC221.Bit 7
            input  Application.a2x4_8 : BOOL  // PLC221.Bit 8
            input  Application.a2x4_9 : BOOL  // PLC221.Bit 9
            input  Application.a2x4_10 : BOOL  // PLC221.Bit 10
            input  Application.a2x4_11 : BOOL  // PLC221.Bit 11
            input  Application.a2x4_12 : BOOL  // PLC221.Bit 12
            input  Application.a2x4_13 : BOOL  // PLC221.Bit 13
            input  Application.a2x4_14 : BOOL  // PLC221.Bit 14
            input  Application.a2x4_15 : BOOL  // PLC221.Bit 15
            input  Application.a2x4_16 : BOOL  // PLC221.Bit 0
            input  Application.a2x4_17 : BOOL  // PLC221.Bit 1
            input  Application.a2x4_18 : BOOL  // PLC221.Bit 2
            input  Application.a2x4_19 : BOOL  // PLC221.Bit 3
            input  Application.a2x4_20 : BOOL  // PLC221.Bit 4
            input  Application.a2x4_21 : BOOL  // PLC221.Bit 5
            input  Application.a2x4_22 : BOOL  // PLC221.Bit 6
            input  Application.a2x4_23 : BOOL  // PLC221.Bit 7
            input  Application.a2x4_24 : BOOL  // PLC221.Bit 8
            input  Application.a2x4_25 : BOOL  // PLC221.Bit 9
            input  Application.a2x4_26 : BOOL  // PLC221.Bit 10
            input  Application.a2x4_27 : BOOL  // PLC221.Bit 11
            input  Application.a2x4_28 : BOOL  // PLC221.Bit 12
            input  Application.a2x4_29 : BOOL  // PLC221.Bit 13
            input  Application.a2x4_30 : BOOL  // PLC221.Bit 14
            input  Application.a2x4_31 : BOOL  // PLC221.Bit 15
            input  Application.a2x5_0 : BOOL  // PLC221.Bit 0
            input  Application.a2x5_1 : BOOL  // PLC221.Bit 1
            input  Application.a2x5_2 : BOOL  // PLC221.Bit 2
            input  Application.a2x5_3 : BOOL  // PLC221.Bit 3
            input  Application.a2x5_4 : BOOL  // PLC221.Bit 4
            input  Application.a2x5_5 : BOOL  // PLC221.Bit 5
            input  Application.a2x5_6 : BOOL  // PLC221.Bit 6
            input  Application.a2x5_7 : BOOL  // PLC221.Bit 7
            input  Application.a2x5_8 : BOOL  // PLC221.Bit 8
            input  Application.a2x5_9 : BOOL  // PLC221.Bit 9
            input  Application.a2x5_10 : BOOL  // PLC221.Bit 10
            input  Application.a2x5_11 : BOOL  // PLC221.Bit 11
            input  Application.a2x5_12 : BOOL  // PLC221.Bit 12
            input  Application.a2x5_13 : BOOL  // PLC221.Bit 13
            input  Application.a2x5_14 : BOOL  // PLC221.Bit 14
            input  Application.a2x5_15 : BOOL  // PLC221.Bit 15
            input  Application.a2x5_16 : BOOL  // PLC221.Bit 0
            input  Application.a2x5_17 : BOOL  // PLC221.Bit 1
            input  Application.a2x5_18 : BOOL  // PLC221.Bit 2
            input  Application.a2x5_19 : BOOL  // PLC221.Bit 3
            input  Application.a2x5_20 : BOOL  // PLC221.Bit 4
            input  Application.a2x5_21 : BOOL  // PLC221.Bit 5
            input  Application.a2x5_22 : BOOL  // PLC221.Bit 6
            input  Application.a2x5_23 : BOOL  // PLC221.Bit 7
            input  Application.a2x5_24 : BOOL  // PLC221.Bit 8
            input  Application.a2x5_25 : BOOL  // PLC221.Bit 9
            input  Application.a2x5_26 : BOOL  // PLC221.Bit 10
            input  Application.a2x5_27 : BOOL  // PLC221.Bit 11
            input  Application.a2x5_28 : BOOL  // PLC221.Bit 12
            input  Application.a2x5_29 : BOOL  // PLC221.Bit 13
            input  Application.a2x5_30 : BOOL  // PLC221.Bit 14
            input  Application.a2x5_31 : BOOL  // PLC221.Bit 15
            input  Application.IW1_0 : WORD  // PLC221
            input  Application.IW1_1 : WORD  // PLC221
            input  Application.IW1_2 : WORD  // PLC221
            input  Application.IW1_3 : WORD  // PLC221
            input  Application.IW2_0 : WORD  // PLC221
            unmapped channels: PLC221, PLC221, PLC221, PLC221, PLC221, PLC221, PLC221, PLC221, PLC221, PLC221, PLC221, PLC221, PLC221, PLC221, PLC221, PLC221, PLC221, PLC221, PLC221, PLC221, PLC221, PLC221, PLC221, PLC221, PLC221
    Serial_Line_1 : Serial line, Schneider Electric, version 4.0.6.18
      Pch : Modbus IOScanner, Schneider Electric, version 3.5.3.8
        PCH_BIG_11_16 : Generic Modbus Slave, Schneider Electric, version 3.5.3.9
            settings: SlaveAddress = 2; ResponseTimeout = 1000; Channel 1.Function Code = 6; Channel 1.Read Offset = 0; Channel 1.Read Length = 0; Channel 1.Write Offset = 16#FA01; Channel 1.Write Length = 1; Channel 1.Cycle Time = 20; Channel 2.Function Code = 3; Channel 2.Read Offset = 16#FD00; Channel 2.Read Length = 1; Channel 2.Write Offset = 0; Channel 2.Write Length = 0; Channel 2.Cycle Time = 100; Channel 3.Function Code = 3; Channel 3.Read Offset = 16#FE03; Channel 3.Read Length = 1; Channel 3.Write Offset = 0; Channel 3.Write Length = 0; Channel 3.Cycle Time = 100
            output WrFreq_pch_big_11_16 : ARRAY[0..0] OF WORD  // Channel 1
            input  ReadFreq_pch_big_11_16 : ARRAY[0..0] OF WORD  // Channel 2
            input  ReadCurr_pch_big_11_16 : ARRAY[0..0] OF WORD  // Channel 3
        PCH_BIG_17_18 : Generic Modbus Slave, Schneider Electric, version 3.5.3.9
            settings: SlaveAddress = 3; ResponseTimeout = 1000; Channel 1.Function Code = 6; Channel 1.Read Offset = 0; Channel 1.Read Length = 0; Channel 1.Write Offset = 16#FA01; Channel 1.Write Length = 1; Channel 1.Cycle Time = 20; Channel 2.Function Code = 3; Channel 2.Read Offset = 16#FD00; Channel 2.Read Length = 1; Channel 2.Write Offset = 0; Channel 2.Write Length = 0; Channel 2.Cycle Time = 100; Channel 3.Function Code = 3; Channel 3.Read Offset = 16#FE03; Channel 3.Read Length = 1; Channel 3.Write Offset = 0; Channel 3.Write Length = 0; Channel 3.Cycle Time = 100
            output WrFreq_pch_big_17_18 : ARRAY[0..0] OF WORD  // Channel 1
            input  ReadFreq_pch_big_17_18 : ARRAY[0..0] OF WORD  // Channel 2
            input  ReadCurr_pch_big_17_18 : ARRAY[0..0] OF WORD  // Channel 3
        PCH_PIT_DROB : Generic Modbus Slave, Schneider Electric, version 3.5.3.9
            settings: SlaveAddress = 1; ResponseTimeout = 1000; Channel 1.Function Code = 6; Channel 1.Read Offset = 0; Channel 1.Read Length = 0; Channel 1.Write Offset = 16#FA01; Channel 1.Write Length = 1; Channel 1.Cycle Time = 20; Channel 2.Function Code = 3; Channel 2.Read Offset = 16#FD00; Channel 2.Read Length = 1; Channel 2.Write Offset = 0; Channel 2.Write Length = 0; Channel 2.Cycle Time = 100; Channel 3.Function Code = 3; Channel 3.Read Offset = 16#FE03; Channel 3.Read Length = 1; Channel 3.Write Offset = 0; Channel 3.Write Length = 0; Channel 3.Cycle Time = 100
            output WrFreq_pch_pit_drob : ARRAY[0..0] OF WORD  // Channel 1
            input  ReadFreq_pch_pit_drob : ARRAY[0..0] OF WORD  // Channel 2
            input  ReadCurr_pch_pit_drob : ARRAY[0..0] OF WORD  // Channel 3
        PCH_MIDLE_201_204 : Generic Modbus Slave, Schneider Electric, version 3.5.3.9
            settings: SlaveAddress = 5; ResponseTimeout = 1000; Channel 1.Function Code = 6; Channel 1.Read Offset = 0; Channel 1.Read Length = 0; Channel 1.Write Offset = 16#FA01; Channel 1.Write Length = 1; Channel 1.Cycle Time = 20; Channel 2.Function Code = 3; Channel 2.Read Offset = 16#FD00; Channel 2.Read Length = 1; Channel 2.Write Offset = 0; Channel 2.Write Length = 0; Channel 2.Cycle Time = 100; Channel 3.Function Code = 3; Channel 3.Read Offset = 16#FE03; Channel 3.Read Length = 1; Channel 3.Write Offset = 0; Channel 3.Write Length = 0; Channel 3.Cycle Time = 100
            output WrFreq_pch_midle_205_209 : ARRAY[0..0] OF WORD  // Channel 1
            input  ReadFreq_pch_midle_205_209 : ARRAY[0..0] OF WORD  // Channel 2
            input  ReadCurr_pch_midle_205_209 : ARRAY[0..0] OF WORD  // Channel 3
        PCH_MIDLE_205_209 : Generic Modbus Slave, Schneider Electric, version 3.5.3.9
            settings: SlaveAddress = 4; ResponseTimeout = 1000; Channel 1.Function Code = 6; Channel 1.Read Offset = 0; Channel 1.Read Length = 0; Channel 1.Write Offset = 16#FA01; Channel 1.Write Length = 1; Channel 1.Cycle Time = 20; Channel 2.Function Code = 3; Channel 2.Read Offset = 16#FD00; Channel 2.Read Length = 1; Channel 2.Write Offset = 0; Channel 2.Write Length = 0; Channel 2.Cycle Time = 100; Channel 3.Function Code = 3; Channel 3.Read Offset = 16#FE03; Channel 3.Read Length = 1; Channel 3.Write Offset = 0; Channel 3.Write Length = 0; Channel 3.Cycle Time = 100
            output WrFreq_pch_midle_201_204 : ARRAY[0..0] OF WORD  // Channel 1
            output qwPCH_MIDLE_201_204_1_Channel_1_0 : WORD  // Channel 1.Channel 1[0]
            input  ReadFreq_pch_midle_201_204 : ARRAY[0..0] OF WORD  // Channel 2
            input  iwPCH_MIDLE_201_204_1_Channel_2_0 : WORD  // Channel 2.Channel 2[0]
            input  ReadCurr_pch_midle_201_204 : ARRAY[0..0] OF WORD  // Channel 3
            input  iwPCH_MIDLE_201_204_1_Channel_3_0 : WORD  // Channel 3.Channel 3[0]
        PCH_SKTR_30330 : Generic Modbus Slave, Schneider Electric, version 3.5.3.9
            settings: SlaveAddress = 7; ResponseTimeout = 1000; Channel 1.Function Code = 6; Channel 1.Read Offset = 0; Channel 1.Read Length = 0; Channel 1.Write Offset = 16#FA01; Channel 1.Write Length = 1; Channel 1.Cycle Time = 20; Channel 2.Function Code = 3; Channel 2.Read Offset = 16#FD00; Channel 2.Read Length = 1; Channel 2.Write Offset = 0; Channel 2.Write Length = 0; Channel 2.Cycle Time = 100; Channel 3.Function Code = 3; Channel 3.Read Offset = 16#FE03; Channel 3.Read Length = 1; Channel 3.Write Offset = 0; Channel 3.Write Length = 0; Channel 3.Cycle Time = 100
            output WrFreq_pch_sktr_30640 : ARRAY[0..0] OF WORD  // Channel 1
            input  ReadFreq_pch_sktr_30640 : ARRAY[0..0] OF WORD  // Channel 2
            input  ReadCurr_pch_sktr_30640 : ARRAY[0..0] OF WORD  // Channel 3
        PCH_SKTR_30640 : Generic Modbus Slave, Schneider Electric, version 3.5.3.9
            settings: SlaveAddress = 6; ResponseTimeout = 1000; Channel 1.Function Code = 6; Channel 1.Read Offset = 0; Channel 1.Read Length = 0; Channel 1.Write Offset = 16#FA01; Channel 1.Write Length = 1; Channel 1.Cycle Time = 20; Channel 2.Function Code = 3; Channel 2.Read Offset = 16#FD00; Channel 2.Read Length = 1; Channel 2.Write Offset = 0; Channel 2.Write Length = 0; Channel 2.Cycle Time = 100; Channel 3.Function Code = 3; Channel 3.Read Offset = 16#FE03; Channel 3.Read Length = 1; Channel 3.Write Offset = 0; Channel 3.Write Length = 0; Channel 3.Cycle Time = 100
            output WrFreq_pch_sktr_30330 : ARRAY[0..0] OF WORD  // Channel 1
            output qwPCH_SKTR_30330_1_Channel_1_0 : WORD  // Channel 1.Channel 1[0]
            input  ReadFreq_pch_sktr_30330 : ARRAY[0..0] OF WORD  // Channel 2
            input  iwPCH_SKTR_30330_1_Channel_2_0 : WORD  // Channel 2.Channel 2[0]
            input  ReadCurr_pch_sktr_30330 : ARRAY[0..0] OF WORD  // Channel 3
            input  iwPCH_SKTR_30330_1_Channel_3_0 : WORD  // Channel 3.Channel 3[0]
    Serial_Line_2 : Serial line, Schneider Electric, version 4.0.6.18
      Weight : Modbus IOScanner, Schneider Electric, version 3.5.3.8
        Weight_Big : Generic Modbus Slave, Schneider Electric, version 3.5.3.9
            settings: SlaveAddress = 1; ResponseTimeout = 500; Channel 1.Function Code = 3; Channel 1.Read Offset = 16#0046; Channel 1.Read Length = 2; Channel 1.Write Offset = 0; Channel 1.Write Length = 0; Channel 1.Cycle Time = 20
            unmapped channels: Channel 1
        Weight_Midle : Generic Modbus Slave, Schneider Electric, version 3.5.3.9
            settings: SlaveAddress = 2; ResponseTimeout = 500; Channel 1.Function Code = 3; Channel 1.Read Offset = 16#0046; Channel 1.Read Length = 2; Channel 1.Write Offset = 0; Channel 1.Write Length = 0; Channel 1.Cycle Time = 20
            unmapped channels: Channel 1
*)

// PLC_241/Application/Real_word
TYPE Real_word :
UNION
	RealValue : REAL;
	WordValue : array[0..1] of word;
END_UNION
END_TYPE

// PLC_241/Application/GVL
VAR_GLOBAL RETAIN
	
	gemer: BOOL;								// глобальная авария
	RESSET AT %MX0.0: BOOL;						// Сброс аварий
	mtune AT %MX0.1: BOOL;						// Ручной режим
	mnaladka AT %MX0.2: BOOL;					// Режим наладки
	mute AT %MX0.3: BOOL;						// Выкл. сирену
	
	write_param_proiz: BOOL;					// Записать параметры производства
	
	PAUSE_BIG_WEIGHT AT %MX0.4: BOOL;			// Паставить на паузу дозирование на больших весах
	PAUSE_MIDLE_WEIGHT AT %MX0.5: BOOL;			// Паставить на паузу дозировние на средних весах
 	Mode_load AT %MX0.6: BOOL;					// Режим загрузки зерновых бункеров
	Mode_load_K AT %MX0.7: BOOL;				// Режим загрузки компонентных бункеров
	Mode_dosing AT %MX0.8: BOOL;				// Режим дозирования на весы 
	Mode_unload AT %MX0.9: BOOL;				// Режим выгрузки готового
	NEW_OTVES AT %MX0.10: BOOL;					// Новый отвес
	TARE_BIG AT %MX0.11: BOOL;					// Учесть тару на больших вессах
	TARE_MIDLE AT %MX0.12: BOOL;				// Учесть тару на средних весах
	RESSET_TARE_BIG_WEIGHT AT %MX0.13: BOOL;	// Сбросить значение тары на 0, большие веса
	RESSET_TARE_MIDLE_WEIGHT AT %MX0.14: BOOL;	// Сбросить значение тары на 0, средние веса
	autoRessetTare_big AT %MX0.15: BOOL;		// Автоматически сбрасывать тару после выгрузки с больших весов
	autoRessetTare_midle AT %MX2.0: BOOL;		// Автоматически сбрасывать тару после выгрузки с средних весов
	
	endQueue AT %MX2.1: BOOL;					// Бит устанавливается со скады что в очереди производства нечего не находиться

// -----------------------------------------------------------------------------------------------------
							// Подсчет порций
// -----------------------------------------------------------------------------------------------------
	one_procent: REAL;			// Вес одного процента от порции  one_procent:= Weight_PORCIA/100.0
	Weight_PORCIA: INT;			// Вес одной порции
	Weight_PATH: INT;			// Общий вес который нужно приготовить
	Tare_big_weight: REAL;		// Вес тары на больших весах
	Tare_midle_weight: REAL;	// Вес тары на средних весах
	OST_BIG_WEIGHT: REAL;		// Остаток на больших весах	(вводиться со скады)
	OST_MIDLE_WEIGHT: REAL;		// Остаток на средних весах	(вводиться со скады)
	
	PORT_NEED: INT;				// количество нужных порций
	PORT_DONE: INT; 			// Приготовленных порций
	PORT_BIG_WEIGHT: WORD;		// Количество сдозированых порций на больших весах
	PORT_SMALL_WEIGHT: INT;		// Количество сдозированых порций на малых весах
	PORD_SMES: INT;				// Количество смешанных порций
	
// -----------------------------------------------------------------------------------------------------

// -----------------------------------------------------------------------------------------------------
							// Блокировка компонента на дозирование в рецепте 
// -----------------------------------------------------------------------------------------------------
	Block_bunk_101 AT %MX4.0: BOOL;
	Block_bunk_102 AT %MX4.1: BOOL;
	Block_bunk_103 AT %MX4.2: BOOL;
	Block_bunk_104 AT %MX4.3: BOOL;
	Block_bunk_105 AT %MX4.4: BOOL;
	Block_bunk_106 AT %MX4.5: BOOL;
	Block_bunk_107 AT %MX4.6: BOOL;
	Block_bunk_108 AT %MX4.7: BOOL;
	Block_bunk_201 AT %MX4.8: BOOL;
	Block_bunk_202 AT %MX4.9: BOOL;
	Block_bunk_203 AT %MX4.10: BOOL;
	Block_bunk_204 AT %MX4.11: BOOL;
	Block_bunk_205 AT %MX4.12: BOOL;
	Block_bunk_206 AT %MX4.13: BOOL;
	Block_bunk_207 AT %MX4.14: BOOL;
	Block_bunk_208 AT %MX4.15: BOOL;
	Block_bunk_209 AT %MX2.2: BOOL;
// -----------------------------------------------------------------------------------------------------


// -----------------------------------------------------------------------------------------------------
							// Использование Дозатора в рецепте
// -----------------------------------------------------------------------------------------------------
	Use_101: BOOL;
	Use_102: BOOL;
	Use_103: BOOL;
	Use_104: BOOL;
	Use_105: BOOL;
	Use_106: BOOL;
	Use_107: BOOL;
	Use_108: BOOL;
	
// -----------------------------------------------------------------------------------------------------

// -----------------------------------------------------------------------------------------------------
							// Переменные по компонентам Больших весов
// -----------------------------------------------------------------------------------------------------
							// Значение (процент компонента в рецепте)
	iKP_101: INT;			// Процент 1 комонента (Вводиться со скады)
		KP_101: REAL;			// Процент 1 комонента (Преобразуется в реал для обработки контроллером)
	iKP_102: INT;			// Процент 2 комонента (Вводиться со скады)
		KP_102: REAL;			// Процент 2 комонента (Преобразуется в реал для обработки контроллером)
	iKP_103: INT;			// Процент 3 комонента (Вводиться со скады)
		KP_103: REAL;			// Процент 3 комонента (Преобразуется в реал для обработки контроллером)
	iKP_104: INT;			// Процент 4 комонента (Вводиться со скады)
		KP_104: REAL;			// Процент 4 комонента (Преобразуется в реал для обработки контроллером)
	iKP_105: INT;			// Процент 5 комонента (Вводиться со скады)
		KP_105: REAL;			// Процент 5 комонента (Преобразуется в реал для обработки контроллером)
	iKP_106: INT;			// Процент 6 комонента (Вводиться со скады)
		KP_106: REAL;			// Процент 6 комонента (Преобразуется в реал для обработки контроллером)
	iKP_107: INT;			// Процент 7 комонента (Вводиться со скады)
		KP_107: REAL;			// Процент 7 комонента (Преобразуется в реал для обработки контроллером)
	iKP_108: INT;			// Процент 8 комонента (Вводиться со скады)
		KP_108: REAL;			// Процент 8 комонента (Преобразуется в реал для обработки контроллером)
		
// -----------------------------------------------------------------------------------------------------

// -----------------------------------------------------------------------------------------------------
							// Значение в кг, масса компонента в рецепте
// -----------------------------------------------------------------------------------------------------
	iK_101: INT;			// Значение для отображения на скаде (Преобразование из реал в инт)
		K_101: REAL;			// Значение реал для обработки контроллером
	iK_102: INT;
		K_102: REAL;
	iK_103: INT;
		K_103: REAL;
	iK_104: INT;
		K_104: REAL;
	iK_105: INT;
		K_105: REAL;
	iK_106: INT;
		K_106: REAL;
	iK_107: INT;
		K_107: REAL;
	iK_108: INT;
		K_108: REAL;
		
// -----------------------------------------------------------------------------------------------------
// -----------------------------------------------------------------------------------------------------
							// Значение выбега 
// -----------------------------------------------------------------------------------------------------
	iFALL_101: INT;			// Значение падающего столба вводимого со скады
		FALL_101: REAL;			// Преобразованное значение падающего столба для обработки контроллером
	iFALL_102: INT;
		FALL_102: REAL;
	iFALL_103: INT;
		FALL_103: REAL;
	iFALL_104: INT;
		FALL_104: REAL;
	iFALL_105: INT;
		FALL_105: REAL;
	iFALL_106: INT;
		FALL_106: REAL;
	iFALL_107: INT;
		FALL_107: REAL;
	iFALL_108: INT;
		FALL_108: REAL;
		
// -----------------------------------------------------------------------------------------------------
							// Новый падающий столб (Выбег) после автоматической коррекции
// -----------------------------------------------------------------------------------------------------
	iNewFall_101: INT;
		NewFall_101: REAL;
	iNewFall_102: INT;
		NewFall_102: REAL;
	iNewFall_103: INT;
		NewFall_103: REAL;
	iNewFall_104: INT;
		NewFall_104: REAL;
	iNewFall_105: INT;
		NewFall_105: REAL;
	iNewFall_106: INT;
		NewFall_106: REAL;
	iNewFall_107: INT;
		NewFall_107: REAL;
	iNewFall_108: INT;
		NewFall_108: REAL;
// -----------------------------------------------------------------------------------------------------

// -----------------------------------------------------------------------------------------------------
							// Биты отвечающик за автоматический расчет падающего столба (Выбега)
// -----------------------------------------------------------------------------------------------------
	autoKorection_101 AT %MX2.3: BOOL:= TRUE;	
	autoKorection_102 AT %MX2.4: BOOL:= TRUE;
	autoKorection_103 AT %MX2.5: BOOL:= TRUE;
	autoKorection_104 AT %MX2.6: BOOL:= TRUE;
	autoKorection_105 AT %MX2.7: BOOL:= TRUE;
	autoKorection_106 AT %MX2.8: BOOL:= TRUE;
	autoKorection_107 AT %MX2.9: BOOL:= TRUE;
	autoKorection_108 AT %MX2.10: BOOL:= TRUE;
	
// -----------------------------------------------------------------------------------------------------
// -----------------------------------------------------------------------------------------------------
							// Значение (Гц) минимальной и максимальной скорости дозирования
// -----------------------------------------------------------------------------------------------------
	vlHISPEED_101: WORD; 	vlLOWSPEED_101: WORD;
	vlHISPEED_102: WORD; 	vlLOWSPEED_102: WORD;
	vlHISPEED_103: WORD; 	vlLOWSPEED_103: WORD;
	vlHISPEED_104: WORD; 	vlLOWSPEED_104: WORD;
	vlHISPEED_105: WORD; 	vlLOWSPEED_105: WORD;
	vlHISPEED_106: WORD; 	vlLOWSPEED_106: WORD;
	vlHISPEED_107: WORD; 	vlLOWSPEED_107: WORD;
	vlHISPEED_108: WORD; 	vlLOWSPEED_108: WORD;
// -----------------------------------------------------------------------------------------------------
	
// -----------------------------------------------------------------------------------------------------
							// Значение (Кг) при котором дазатор начинает снижать скорость дозирования для точного дозирования на весы
// -----------------------------------------------------------------------------------------------------
	ivlDropSpeed_101: INT;	vlDropSpeed_101: REAL;
	ivlDropSpeed_102: INT;	vlDropSpeed_102: REAL;
	ivlDropSpeed_103: INT;	vlDropSpeed_103: REAL;
	ivlDropSpeed_104: INT;	vlDropSpeed_104: REAL;
	ivlDropSpeed_105: INT;	vlDropSpeed_105: REAL;
	ivlDropSpeed_106: INT;	vlDropSpeed_106: REAL;
	ivlDropSpeed_107: INT;	vlDropSpeed_107: REAL;
	ivlDropSpeed_108: INT;	vlDropSpeed_108: REAL;
// -----------------------------------------------------------------------------------------------------
	
// -----------------------------------------------------------------------------------------------------
							// Значение (%) допустимое отклонение	+/-	
// -----------------------------------------------------------------------------------------------------
	ivlPlusDeviation_101: INT; 	ivlMinusDeviation_101: INT;
	ivlPlusDeviation_102: INT; 	ivlMinusDeviation_102: INT;
	ivlPlusDeviation_103: INT; 	ivlMinusDeviation_103: INT;
	ivlPlusDeviation_104: INT;	ivlMinusDeviation_104: INT;
	ivlPlusDeviation_105: INT; 	ivlMinusDeviation_105: INT;
	ivlPlusDeviation_106: INT; 	ivlMinusDeviation_106: INT;
	ivlPlusDeviation_107: INT;	ivlMinusDeviation_107: INT;
	ivlPlusDeviation_108: INT;	ivlMinusDeviation_108: INT;
	
// -----------------------------------------------------------------------------------------------------
							// Значение (кг) допустимое отклонение	+/-	каждого компонента
// -----------------------------------------------------------------------------------------------------
	vlPlusDeviation_101: REAL;	vlMinusDeviation_101: REAL;
	vlPlusDeviation_102: REAL;	vlMinusDeviation_102: REAL;
	vlPlusDeviation_103: REAL;	vlMinusDeviation_103: REAL;
	vlPlusDeviation_104: REAL;	vlMinusDeviation_104: REAL;
	vlPlusDeviation_105: REAL;	vlMinusDeviation_105: REAL;
	vlPlusDeviation_106: REAL;	vlMinusDeviation_106: REAL;
	vlPlusDeviation_107: REAL;	vlMinusDeviation_107: REAL;
	vlPlusDeviation_108: REAL;	vlMinusDeviation_108: REAL;
// -----------------------------------------------------------------------------------------------------
	
	

// -----------------------------------------------------------------------------------------------------

// -----------------------------------------------------------------------------------------------------
				// Дозирование на веса
// -----------------------------------------------------------------------------------------------------
	array_dosing_Z AT %MW1200: ARRAY[1..9] OF WORD;		// Массив очереди дозирования больших весов (в ячейке храниться номер бункера из которого нужно дозировать)
	STEP_Z: WORD:= 1;									// Стетчик для массива очереди дозирования больших вессов
	array_dozing_K AT %MW1300: ARRAY[1..10] OF WORD;	// Массив очереди дозирования средних весов (в ячейке храниться номер бункера из которого нужно дозировать)
	STEP_K: WORD;										// Стетчик для массива очереди дозирования средних вессов
// -----------------------------------------------------------------------------------------------------

	use_scalp AT %MX2.13: BOOL;			// Использование скальператора 
	
// -----------------------------------------------------------------------------------------------------
				// Параметр устанавливается из скады для выбора бункера в который грузиться сырье
// -----------------------------------------------------------------------------------------------------
	numberBunkAddWeight_Z AT %MW2000: INT; 	// Храниться номер бункера для дабавления или удаления значения текущего весса в ручную... Сырье 
	numberBunkAddWeight_K AT %MW2002: INT; 	// Храниться номер бункера для дабавления или удаления значения текущего весса в ручную... Добавки
	AddWeight AT %MD2004: REAL; 			// Значение дабавляемого весса в бункер
	AddLoad_weight AT %MX2.11: BOOL;		// Бит отвечающий за дабавление весса в бункер
	DeleteLoad_weight AT %MX2.12: BOOL;		// Бит отвечающий за удаление весса из бункера

// -----------------------------------------------------------------------------------------------------	
	
// -----------------------------------------------------------------------------------------------------	
								// Зерновые бункера
// -----------------------------------------------------------------------------------------------------	
	array_load_queue AT %MW1000: ARRAY[1..9] OF WORD; 	// Массив очереди загрузки зерновых бункеров
	array_load_K_queue AT %MW1100: ARRAY[1..5] OF WORD;	// Массив очереди загрузки компонентов
	currItem_queue AT %MW6032: WORD;					// Текущий бункер для загрузки в очереди
	nextItem_queue AT %MW6033: WORD;					// Следующий бункер для загрузки в очереди
	currItem_queue_K AT %MW6034: WORD;					// Текущий бункер для загрузки в очереди компонентов
	nextItem_queue_K AT %MW6035: WORD;					// Следующий бункер для загрузки в очереди компонентов
	btnNext_load_Z AT %MX2.15: BOOL;					// Переход к следующему бункеру в очереди (Загрузка сырья)
	btnNext_load_K AT %MX100.0: BOOL;					// Переход к следующему бункеру в очереди (Загрузка Компонентов)	
	timePause_load_queue AT %MW5999: WORD;				// пауза между загрузкой, время на очистку оборудования в линии
	timePause_load_K_queue AT %MW5998: WORD;			// пауза между загрузкой компонентов, время на очистку оборудования в линии 
	
	timePause_DNY_HOLE AT %MW5997: WORD;				// пауза для отключения режима "Загрузка зерновых бункеров" при пустой яме
	use_time_hole AT %MX2.14: BOOL;						// Использования функции авто выключения режима по датчику в завальной яме
	
// -----------------------------------------------------------------------------------------------------	
										// текущий вес в зерновых бункерах
// -----------------------------------------------------------------------------------------------------	
	currWeight_bunk_101 AT %MD6000: REAL;
	currWeight_bunk_102 AT %MD6002: REAL;
	currWeight_bunk_103 AT %MD6004: REAL;
	currWeight_bunk_104 AT %MD6006: REAL;
	currWeight_bunk_105 AT %MD6008: REAL;
	currWeight_bunk_106 AT %MD6010: REAL;
	currWeight_bunk_107 AT %MD6012: REAL;
	currWeight_bunk_108 AT %MD6014: REAL;
// -----------------------------------------------------------------------------------------------------	
// -----------------------------------------------------------------------------------------------------	
										// текущий вес в бункерах компонентов
// -----------------------------------------------------------------------------------------------------
	currWeight_bunk_201 AT %MD6016: REAL;
	currWeight_bunk_202 AT %MD6018: REAL;
	currWeight_bunk_203 AT %MD6020: REAL;
	currWeight_bunk_204 AT %MD6022: REAL;
	currWeight_bunk_205 AT %MD6024: REAL;
	currWeight_bunk_206 AT %MD6026: REAL;
	currWeight_bunk_207 AT %MD6028: REAL;
	currWeight_bunk_208 AT %MD6030: REAL;
	currWeight_bunk_209 AT %MD6032: REAL;
// -----------------------------------------------------------------------------------------------------
	
//---------------------------------------------------------------------------------------------------------------------------
										// Временные задержки для датчиков и механизмов
//---------------------------------------------------------------------------------------------------------------------------
	// Конвейер завальной ямы
		TimeStart_SKTR_10110 AT %MW8000: WORD;
		TimeStop_SKTR_10110 AT %MW8001: WORD;
		TimeDP_SKTR_10110 AT %MW8002: WORD;
	
	// Локальный фильтр нории 10200 (АС 10201)
		TimeStart_Localfilter_10201 AT %MW8003: WORD;
		TimeStop_Localfilter_10201 AT %MW8004: WORD;
		
	// Нория 10200
		TimeStart_noria_10200 AT %MW8005: WORD;
		TimeStop_noria_10200 AT %MW8006: WORD;
		TimeDKS_noria_10200 AT %MW8007: WORD;
		TimeDSL_noria_10200 AT %MW8008: WORD;
		TimeDP_noria_10200 AT %MW8009: WORD;
		
	// Нория 10400
		TimeStart_noria_10400 AT %MW8010: WORD;
		TimeStop_noria_10400 AT %MW8011: WORD;
		TimeDKS_noria_10400 AT %MW8012: WORD;
		TimeDSL_noria_10400 AT %MW8013: WORD;
		TimeDP_noria_10400 AT %MW8014: WORD;
		
	// Нория 21200
		TimeStart_noria_21200 AT %MW8015: WORD;
		TimeStop_noria_21200 AT %MW8016: WORD;
		TimeDKS_noria_21200 AT %MW8017: WORD;
		TimeDSL_noria_21200 AT %MW8018: WORD;
		TimeDP_noria_21200 AT %MW8019: WORD;
		
	// 2-х ходовая заслонка 10210
		TimeLT_flap_10210 AT %MW8020: WORD;
		TimePol_scalp_flap_10210 AT %MW8021: WORD;
		TimePol_noria_flap_10210 AT %MW8022: WORD;
		
	// Скальператор
		TimeStart_scalp AT %MW8023: WORD;
		TimeStop_scalp AT %MW8024: WORD;
	
	// Локальный фильтр нории 10400 (АС 10401)
		TimeStart_Localfilter_10401 AT %MW8025: WORD;
		TimeStop_Localfilter_10401 AT %MW8026: WORD;
	
	// Локальный фильтр Конвейера 10500 (АС 10501)
		TimeStart_Localfilter_10501 AT %MW8027: WORD;
		TimeStop_Localfilter_10501 AT %MW8028: WORD;
		
	//Конвейер 10500
		TimeStart_SKTR_10500 AT %MW8029: WORD;
		TimeStop_SKTR_10500 AT %MW8030: WORD;
		TimeDKS_SKTR_10500 AT %MW8031: WORD;
		TimeDP_SKTR_10500 AT %MW8032: WORD;
		
	// 2-х ходовая заслонка 10710
		timeLT_tflap_10710 AT %MW8033: WORD;
		timePol_1_tflap_10710 AT %MW8034: WORD;
		timePol_2_tflap_10710 AT %MW8035: WORD;
		
	// Шибер 10610 конвейера 10500
		timeLT_sh_10610 AT %MW8036: WORD;
		timeOpen_sh_10610 AT %MW8037: WORD;
		timeClose_sh_10610 AT %MW8038: WORD;
		
	// 2-х ходовая заслонка 10720
		timeLT_tflap_10720 AT %MW8039: WORD;
		timePol_1_tflap_10720 AT %MW8040: WORD;
		timePol_2_tflap_10720 AT %MW8041: WORD;
		
	// Шибер 10620 конвейера 10500
		timeLT_sh_10620 AT %MW8042: WORD;
		timeOpen_sh_10620 AT %MW8043: WORD;
		timeClose_sh_10620 AT %MW8044: WORD;
		
	// 2-х ходовая заслонка 10730
		timeLT_tflap_10730 AT %MW8045: WORD;
		timePol_1_tflap_10730 AT %MW8046: WORD;
		timePol_2_tflap_10730 AT %MW8047: WORD;
		
	// Шибер 10630 конвейера 10500
		timeLT_sh_10630 AT %MW8048: WORD;
		timeOpen_sh_10630 AT %MW8049: WORD;
		timeClose_sh_10630 AT %MW8050: WORD;
		
	// 2-х ходовая заслонка 10740
		timeLT_tflap_10740 AT %MW8051: WORD;
		timePol_1_tflap_10740 AT %MW8052: WORD;
		timePol_2_tflap_10740 AT %MW8053: WORD;
		
	// Шибер 10640 конвейера 10500
		timeLT_sh_10640 AT %MW8054: WORD;
		timeOpen_sh_10640 AT %MW8055: WORD;
		timeClose_sh_10640 AT %MW8056: WORD;
		
	// Шибер 21310 конвейера 21300
		timeLT_sh_21310 AT %MW8057: WORD;
		timeOpen_sh_21310 AT %MW8058: WORD;
		timeClose_sh_21310 AT %MW8059: WORD;
		
	// Шибер 21320 конвейера 21300
		timeLT_sh_21320 AT %MW8060: WORD;
		timeOpen_sh_21320 AT %MW8061: WORD;
		timeClose_sh_21320 AT %MW8062: WORD;
		
	// Шибер 21330 конвейера 21300
		timeLT_sh_21330 AT %MW8063: WORD;
		timeOpen_sh_21330 AT %MW8064: WORD;
		timeClose_sh_21330 AT %MW8065: WORD;
		
	// Фильтр-шкаф на завальной яме
		timeStart_fans_hole AT %MW8066: WORD;
		timeStop_fans_hole AT %MW8067: WORD;
		
	// Шнек 21300
		timeDKS_shnek_21300 AT %MW8068: WORD;
		timeDP_shnek_21300 AT %MW8069: WORD;
		timeStart_shnek_21300 AT %MW8070: WORD;
		timeStop_shnek_21300 AT %MW8071: WORD;
		
	// Шнек 20011
		timeDP_doz_shnek_20011 AT %MW8072: WORD;
		timeStart_doz_shnek_20011 AT %MW8073: WORD;
	// Шнек 20012
		timeDP_doz_shnek_20012 AT %MW8074: WORD;
		timeStart_doz_shnek_20012 AT %MW8075: WORD;
	// Шнек 20013
		timeDP_doz_shnek_20013 AT %MW8076: WORD;
		timeStart_doz_shnek_20013 AT %MW8077: WORD;
	// Шнек 20014
		timeDP_doz_shnek_20014 AT %MW8078: WORD;
		timeStart_doz_shnek_20014 AT %MW8079: WORD;
	// Шнек 20015
		timeDP_doz_shnek_20015 AT %MW8080: WORD;
		timeStart_doz_shnek_20015 AT %MW8081: WORD;
	// Шнек 20016
		timeDP_doz_shnek_20016 AT %MW8082: WORD;
		timeStart_doz_shnek_20016 AT %MW8083: WORD;
	// Шнек 20017
		timeDP_doz_shnek_20017 AT %MW8084: WORD;
		timeStart_doz_shnek_20017 AT %MW8085: WORD;
	// Шнек 20018
		timeDP_doz_shnek_20018 AT %MW8086: WORD;
		timeStart_doz_shnek_20018 AT %MW8088: WORD;
	
	// Шнек 20110
		timeDKS_sktr_20110 AT %MW8089: WORD;
		timeDP_sktr_20110 AT %MW8090: WORD;
		timeStart_sktr_20110 AT %MW8091: WORD;
		timeStop_sktr_20110 AT %MW8092: WORD;
		
	// Датчики уровня
		timeDVY_load AT %MW8093: WORD;
		timeDNU_load AT %MW8094: WORD;
// -----------------------------------------------------------------------------------------------------
	
	
// -----------------------------------------------------------------------------------------------------
							// Отключение датчиков из скады
// -----------------------------------------------------------------------------------------------------
	// Конвейер завальной ямы
		offDP_SKTR_10110 AT %MX6.0: BOOL;
	
	// Нория 10200
		offdks_noria_10200 AT %MX6.1: BOOL;
		offdsl1_noria_10200 AT %MX6.2: BOOL;
		offdsl2_noria_10200 AT %MX6.3: BOOL;
		offdp_noria_10200 AT %MX6.4: BOOL;
	
	// Нория 10400
		offdks_noria_10400 AT %MX6.5: BOOL;
		offdsl1_noria_10400 AT %MX6.6: BOOL;
		offdsl2_noria_10400 AT %MX6.7: BOOL;
		offdp_noria_10400 AT %MX6.8: BOOL;
	
	// Нория 21200
		offdks_noria_21200 AT %MX6.9: BOOL;
		offdsl1_noria_21200 AT %MX6.10: BOOL;
		offdsl2_noria_21200 AT %MX6.11: BOOL;
		offdp_noria_21200 AT %MX6.12: BOOL;
		
	// Конвейер 10500
		offDKS_SKTR_10500 AT %MX6.13: BOOL;
		offDP_SKTR_10500 AT %MX6.14: BOOL;
		
	// Шнек 21300
		offDKS_shnek_21300 AT %MX6.15: BOOL;
		offDP_shnek_21300 AT %MX8.0: BOOL;
		
	// Дозирующий шнек 20011
		offDP_doz_shnek_20011 AT %MX8.1: BOOL;
	// Дозирующий шнек 20012
		offDP_doz_shnek_20012 AT %MX8.2: BOOL;
	// Дозирующий шнек 20013
		offDP_doz_shnek_20013 AT %MX8.3: BOOL;
	// Дозирующий шнек 20014
		offDP_doz_shnek_20014 AT %MX8.4: BOOL;
	// Дозирующий шнек 20015
		offDP_doz_shnek_20015 AT %MX8.5: BOOL;
	// Дозирующий шнек 20016
		offDP_doz_shnek_20016 AT %MX8.6: BOOL;
	// Дозирующий шнек 20017
		offDP_doz_shnek_20017 AT %MX8.7: BOOL;
	// Дозирующий шнек 20018
		offDP_doz_shnek_20018 AT %MX8.8: BOOL;
		
	// конвейер выгрубной под большими весами 20110
		offDKS_sktr_20110 AT %MX8.9: BOOL;
		offDP_sktr_20110 AT %MX8.10: BOOL;
		
	
// -----------------------------------------------------------------------------------------------------
							// Наработка моточасов на оборудовании
// -----------------------------------------------------------------------------------------------------
	MH_sktr_10110 AT %MD7000: DINT;
	MH_AC_1_1 AT %MD7002: DINT;
	MH_AC_1_2 AT %MD7004: DINT;
	MH_Noria_10200 AT %MD7006: DINT;
	MH_LF_Noria_10200 AT %MD7008: DINT;
	MH_Scalp AT %MD7010: DINT;
	MH_Noria_10400 AT %MD7012: DINT;
	MH_LF_Noria_10400 AT %MD7014: DINT;
	MH_sktr_10500 AT %MD7016: DINT;
	MH_LF_sktr_10500 AT %MD7018: DINT;
	MH_SH_10610 AT %MD7020: DINT;
	MH_SH_10620 AT %MD7022: DINT;
	MH_SH_10630 AT %MD7024: DINT;
	MH_SH_10640 AT %MD7026: DINT;
	MH_doz_shnek_20011 AT %MD7028: DINT;
	MH_doz_shnek_20012 AT %MD7030: DINT;
	MH_doz_shnek_20013 AT %MD7032: DINT;
	MH_doz_shnek_20014 AT %MD7034: DINT;
	MH_doz_shnek_20015 AT %MD7036: DINT;
	MH_doz_shnek_20016 AT %MD7038: DINT;
	MH_doz_shnek_20017 AT %MD7040: DINT;
	MH_doz_shnek_20018 AT %MD7042: DINT;
	MH_sktr_20110 AT %MD7044: DINT;
	MH_Noria_20300 AT %MD7046: DINT;
	MH_LF_Noria_20301 AT %MD7048: DINT;
	MH_SH_30110 AT %MD7050: DINT;
	MH_doz_pit_drob AT %MD7052: DINT;
	MH_drob AT %MD7054: DINT;
	MH_shnek_30330 AT %MD7056: DINT;
	MH_shluz_30340 AT %MD7058: DINT;
	MH_asp_drob_30310 AT %MD7060: DINT;
	MH_sktr_30400 AT %MD7062: DINT;
	MH_Noria_21200 AT %MD7064: DINT;
	MH_shnek_21300 AT %MD7066: DINT;
	MH_SH_21310 AT %MD7068: DINT;
	MH_SH_21320 AT %MD7070: DINT;
	MH_SH_21330 AT %MD7072: DINT;
	MH_doz_shnek_21410 AT %MD7074: DINT;
	MH_doz_shnek_21411 AT %MD7076: DINT;
	MH_doz_shnek_21412 AT %MD7078: DINT;
	MH_doz_shnek_21413 AT %MD7080: DINT;
	MH_doz_shnek_21414 AT %MD7082: DINT;
	MH_doz_shnek_21510 AT %MD7086: DINT;
	MH_doz_shnek_21520 AT %MD7088: DINT;
	MH_doz_shnek_21530 AT %MD7090: DINT;
	MH_doz_shnek_21540 AT %MD7092: DINT;
	MH_shnek_21600 AT %MD7094: DINT;
	MH_Noria_30500 AT %MD7096: DINT;
	MH_Smes AT %MD7098: DINT;
	MH_shnek_30640 AT %MD7100: DINT;
	MH_Noria_30700 AT %MD7102: DINT;
	MH_LF_Noria_30700 AT %MD7104: DINT;
	MH_sktr_30900 AT %MD7106: DINT;
	MH_LF_sktr_30900 AT %MD7108: DINT;
	MH_SH_30910 AT %MD7110: DINT;
	MH_SH_30920 AT %MD7112: DINT;
	MH_SH_30930 AT %MD7114: DINT;
	MH_SH_30940 AT %MD7116: DINT;
	MH_sktr_30800 AT %MD7118: DINT;
	MH_SH_30810 AT %MD7120: DINT;
	MH_SH_30820 AT %MD7122: DINT;
	MH_KP_10210 AT %MD7124: DINT;
	MH_KP_10710 AT %MD7126: DINT;
	MH_KP_10720 AT %MD7128: DINT;
	MH_KP_10730 AT %MD7130: DINT;
	MH_KP_10740 AT %MD7132: DINT;
// -----------------------------------------------------------------------------------------------------
	
	
	
END_VAR

// PLC_241/Application/IN_OUT
VAR_GLOBAL
	x0_0: BOOL;
	x0_1: BOOL;
	x0_2: BOOL;
	x0_3: BOOL;
	x0_4: BOOL;
	x0_5: BOOL;
	x0_6: BOOL;
	x0_7: BOOL;
	x0_8: BOOL;
	x0_9: BOOL;
	x0_10: BOOL;
	x0_11: BOOL;
	x0_12: BOOL;
	x0_13: BOOL;
	x0_14: BOOL;
	x0_15: BOOL;
	x0_16: BOOL;
	x0_17: BOOL;
	x0_18: BOOL;
	x0_19: BOOL;
	x0_20: BOOL;
	x0_21: BOOL;
	x0_22: BOOL;
	x0_23: BOOL;
	
	y0_0: BOOL;
	y0_1: BOOL;
	y0_2: BOOL;
	y0_3: BOOL;
	y0_4: BOOL;
	y0_5: BOOL;
	y0_6: BOOL;
	y0_7: BOOL;
	y0_8: BOOL;
	y0_9: BOOL;
	y0_10: BOOL;
	y0_11: BOOL;
	y0_12: BOOL;
	y0_13: BOOL;
	y0_14: BOOL;
	y0_15: BOOL;
	
	x1_0: BOOL;
	x1_1: BOOL;
	x1_2: BOOL;
	x1_3: BOOL;
	x1_4: BOOL;
	x1_5: BOOL;
	x1_6: BOOL;
	x1_7: BOOL;
	x1_8: BOOL;
	x1_9: BOOL;
	x1_10: BOOL;
	x1_11: BOOL;
	x1_12: BOOL;
	x1_13: BOOL;
	x1_14: BOOL;
	x1_15: BOOL;
	x1_16: BOOL;
	x1_17: BOOL;
	x1_18: BOOL;
	x1_19: BOOL;
	x1_20: BOOL;
	x1_21: BOOL;
	x1_22: BOOL;
	x1_23: BOOL;
	x1_24: BOOL;
	x1_25: BOOL;
	x1_26: BOOL;
	x1_27: BOOL;
	x1_28: BOOL;
	x1_29: BOOL;
	x1_30: BOOL;
	x1_31: BOOL;
	
	x2_0: BOOL;
	x2_1: BOOL;
	x2_2: BOOL;
	x2_3: BOOL;
	x2_4: BOOL;
	x2_5: BOOL;
	x2_6: BOOL;
	x2_7: BOOL;
	x2_8: BOOL;
	x2_9: BOOL;
	x2_10: BOOL;
	x2_11: BOOL;
	x2_12: BOOL;
	x2_13: BOOL;
	x2_14: BOOL;
	x2_15: BOOL;
	x2_16: BOOL;
	x2_17: BOOL;
	x2_18: BOOL;
	x2_19: BOOL;
	x2_20: BOOL;
	x2_21: BOOL;
	x2_22: BOOL;
	x2_23: BOOL;
	x2_24: BOOL;
	x2_25: BOOL;
	x2_26: BOOL;
	x2_27: BOOL;
	x2_28: BOOL;
	x2_29: BOOL;
	x2_30: BOOL;
	x2_31: BOOL;
	
	x3_0: BOOL;
	x3_1: BOOL;
	x3_2: BOOL;
	x3_3: BOOL;
	x3_4: BOOL;
	x3_5: BOOL;
	x3_6: BOOL;
	x3_7: BOOL;
	x3_8: BOOL;
	x3_9: BOOL;
	x3_10: BOOL;
	x3_11: BOOL;
	x3_12: BOOL;
	x3_13: BOOL;
	x3_14: BOOL;
	x3_15: BOOL;
	x3_16: BOOL;
	x3_17: BOOL;
	x3_18: BOOL;
	x3_19: BOOL;
	x3_20: BOOL;
	x3_21: BOOL;
	x3_22: BOOL;
	x3_23: BOOL;
	x3_24: BOOL;
	x3_25: BOOL;
	x3_26: BOOL;
	x3_27: BOOL;
	x3_28: BOOL;
	x3_29: BOOL;
	x3_30: BOOL;
	x3_31: BOOL;
	
	x4_0: BOOL;
	x4_1: BOOL;
	x4_2: BOOL;
	x4_3: BOOL;
	x4_4: BOOL;
	x4_5: BOOL;
	x4_6: BOOL;
	x4_7: BOOL;
	x4_8: BOOL;
	x4_9: BOOL;
	x4_10: BOOL;
	x4_11: BOOL;
	x4_12: BOOL;
	x4_13: BOOL;
	x4_14: BOOL;
	x4_15: BOOL;
	x4_16: BOOL;
	x4_17: BOOL;
	x4_18: BOOL;
	x4_19: BOOL;
	x4_20: BOOL;
	x4_21: BOOL;
	x4_22: BOOL;
	x4_23: BOOL;
	x4_24: BOOL;
	x4_25: BOOL;
	x4_26: BOOL;
	x4_27: BOOL;
	x4_28: BOOL;
	x4_29: BOOL;
	x4_30: BOOL;
	x4_31: BOOL;
	
	x5_0: BOOL;
	x5_1: BOOL;
	x5_2: BOOL;
	x5_3: BOOL;
	x5_4: BOOL;
	x5_5: BOOL;
	x5_6: BOOL;
	x5_7: BOOL;
	x5_8: BOOL;
	x5_9: BOOL;
	x5_10: BOOL;
	x5_11: BOOL;
	x5_12: BOOL;
	x5_13: BOOL;
	x5_14: BOOL;
	x5_15: BOOL;
	x5_16: BOOL;
	x5_17: BOOL;
	x5_18: BOOL;
	x5_19: BOOL;
	x5_20: BOOL;
	x5_21: BOOL;
	x5_22: BOOL;
	x5_23: BOOL;
	x5_24: BOOL;
	x5_25: BOOL;
	x5_26: BOOL;
	x5_27: BOOL;
	x5_28: BOOL;
	x5_29: BOOL;
	x5_30: BOOL;
	x5_31: BOOL;
	
	y6_0: BOOL;
	y6_1: BOOL;
	y6_2: BOOL;
	y6_3: BOOL;
	y6_4: BOOL;
	y6_5: BOOL;
	y6_6: BOOL;
	y6_7: BOOL;
	y6_8: BOOL;
	y6_9: BOOL;
	y6_10: BOOL;
	y6_11: BOOL;
	y6_12: BOOL;
	y6_13: BOOL;
	y6_14: BOOL;
	y6_15: BOOL;
	y6_16: BOOL;
	y6_17: BOOL;
	y6_18: BOOL;
	y6_19: BOOL;
	y6_20: BOOL;
	y6_21: BOOL;
	y6_22: BOOL;
	y6_23: BOOL;
	y6_24: BOOL;
	y6_25: BOOL;
	y6_26: BOOL;
	y6_27: BOOL;
	y6_28: BOOL;
	y6_29: BOOL;
	y6_30: BOOL;
	y6_31: BOOL;
	
	y7_0: BOOL;
	y7_1: BOOL;
	y7_2: BOOL;
	y7_3: BOOL;
	y7_4: BOOL;
	y7_5: BOOL;
	y7_6: BOOL;
	y7_7: BOOL;
	y7_8: BOOL;
	y7_9: BOOL;
	y7_10: BOOL;
	y7_11: BOOL;
	y7_12: BOOL;
	y7_13: BOOL;
	y7_14: BOOL;
	y7_15: BOOL;
	y7_16: BOOL;
	y7_17: BOOL;
	y7_18: BOOL;
	y7_19: BOOL;
	y7_20: BOOL;
	y7_21: BOOL;
	y7_22: BOOL;
	y7_23: BOOL;
	y7_24: BOOL;
	y7_25: BOOL;
	y7_26: BOOL;
	y7_27: BOOL;
	y7_28: BOOL;
	y7_29: BOOL;
	y7_30: BOOL;
	y7_31: BOOL;
	
	a2x0_0: BOOL;
	a2x0_1: BOOL;
	a2x0_2: BOOL;
	a2x0_3: BOOL;
	a2x0_4: BOOL;
	a2x0_5: BOOL;
	a2x0_6: BOOL;
	a2x0_7: BOOL;
	a2x0_8: BOOL;
	a2x0_9: BOOL;
	a2x0_10: BOOL;
	a2x0_11: BOOL;
	a2x0_12: BOOL;
	a2x0_13: BOOL;
	a2x0_14: BOOL;
	a2x0_15: BOOL;
	a2x0_16: BOOL;
	a2x0_17: BOOL;
	a2x0_18: BOOL;
	a2x0_19: BOOL;
	a2x0_20: BOOL;
	a2x0_21: BOOL;
	a2x0_22: BOOL;
	a2x0_23: BOOL;
	
	a2y0_0: BOOL;
	a2y0_1: BOOL;
	a2y0_2: BOOL;
	a2y0_3: BOOL;
	a2y0_4: BOOL;
	a2y0_5: BOOL;
	a2y0_6: BOOL;
	a2y0_7: BOOL;
	a2y0_8: BOOL;
	a2y0_9: BOOL;
	a2y0_10: BOOL;
	a2y0_11: BOOL;
	a2y0_12: BOOL;
	a2y0_13: BOOL;
	a2y0_14: BOOL;
	a2y0_15: BOOL;
	
	a2x3_0: BOOL;
	a2x3_1: BOOL;
	a2x3_2: BOOL;
	a2x3_3: BOOL;
	a2x3_4: BOOL;
	a2x3_5: BOOL;
	a2x3_6: BOOL;
	a2x3_7: BOOL;
	a2x3_8: BOOL;
	a2x3_9: BOOL;
	a2x3_10: BOOL;
	a2x3_11: BOOL;
	a2x3_12: BOOL;
	a2x3_13: BOOL;
	a2x3_14: BOOL;
	a2x3_15: BOOL;
	a2x3_16: BOOL;
	a2x3_17: BOOL;
	a2x3_18: BOOL;
	a2x3_19: BOOL;
	a2x3_20: BOOL;
	a2x3_21: BOOL;
	a2x3_22: BOOL;
	a2x3_23: BOOL;
	a2x3_24: BOOL;
	a2x3_25: BOOL;
	a2x3_26: BOOL;
	a2x3_27: BOOL;
	a2x3_28: BOOL;
	a2x3_29: BOOL;
	a2x3_30: BOOL;
	a2x3_31: BOOL;
	
	a2x4_0: BOOL;
	a2x4_1: BOOL;
	a2x4_2: BOOL;
	a2x4_3: BOOL;
	a2x4_4: BOOL;
	a2x4_5: BOOL;
	a2x4_6: BOOL;
	a2x4_7: BOOL;
	a2x4_8: BOOL;
	a2x4_9: BOOL;
	a2x4_10: BOOL;
	a2x4_11: BOOL;
	a2x4_12: BOOL;
	a2x4_13: BOOL;
	a2x4_14: BOOL;
	a2x4_15: BOOL;
	a2x4_16: BOOL;
	a2x4_17: BOOL;
	a2x4_18: BOOL;
	a2x4_19: BOOL;
	a2x4_20: BOOL;
	a2x4_21: BOOL;
	a2x4_22: BOOL;
	a2x4_23: BOOL;
	a2x4_24: BOOL;
	a2x4_25: BOOL;
	a2x4_26: BOOL;
	a2x4_27: BOOL;
	a2x4_28: BOOL;
	a2x4_29: BOOL;
	a2x4_30: BOOL;
	a2x4_31: BOOL;
	
	a2x5_0: BOOL;
	a2x5_1: BOOL;
	a2x5_2: BOOL;
	a2x5_3: BOOL;
	a2x5_4: BOOL;
	a2x5_5: BOOL;
	a2x5_6: BOOL;
	a2x5_7: BOOL;
	a2x5_8: BOOL;
	a2x5_9: BOOL;
	a2x5_10: BOOL;
	a2x5_11: BOOL;
	a2x5_12: BOOL;
	a2x5_13: BOOL;
	a2x5_14: BOOL;
	a2x5_15: BOOL;
	a2x5_16: BOOL;
	a2x5_17: BOOL;
	a2x5_18: BOOL;
	a2x5_19: BOOL;
	a2x5_20: BOOL;
	a2x5_21: BOOL;
	a2x5_22: BOOL;
	a2x5_23: BOOL;
	a2x5_24: BOOL;
	a2x5_25: BOOL;
	a2x5_26: BOOL;
	a2x5_27: BOOL;
	a2x5_28: BOOL;
	a2x5_29: BOOL;
	a2x5_30: BOOL;
	a2x5_31: BOOL;
	
	a2y6_0: BOOL;
	a2y6_1: BOOL;
	a2y6_2: BOOL;
	a2y6_3: BOOL;
	a2y6_4: BOOL;
	a2y6_5: BOOL;
	a2y6_6: BOOL;
	a2y6_7: BOOL;
	a2y6_8: BOOL;
	a2y6_9: BOOL;
	a2y6_10: BOOL;
	a2y6_11: BOOL;
	a2y6_12: BOOL;
	a2y6_13: BOOL;
	a2y6_14: BOOL;
	a2y6_15: BOOL;
	a2y6_16: BOOL;
	a2y6_17: BOOL;
	a2y6_18: BOOL;
	a2y6_19: BOOL;
	a2y6_20: BOOL;
	a2y6_21: BOOL;
	a2y6_22: BOOL;
	a2y6_23: BOOL;
	a2y6_24: BOOL;
	a2y6_25: BOOL;
	a2y6_26: BOOL;
	a2y6_27: BOOL;
	a2y6_28: BOOL;
	a2y6_30: BOOL;
	a2y6_31: BOOL;
	
	IW1_0: WORD;
	IW1_1: WORD;
	IW1_2: WORD;
	IW1_3: WORD;
	
	IW2_0: WORD;
END_VAR

// PLC_241/Application/Mechanizm
VAR_GLOBAL
	errbtnpusk: BOOL;
	emerstop_shu: BOOL;
	emerstop_scalp: BOOL;
	emerstop_drob: BOOL;
	emerstop_smes: BOOL;
	emerstop_ubload_bunk: BOOL;
	errrkf: BOOL;
	
	run_sirena: BOOL;
	run_alarm: BOOL;
	
// Конвейер скребковый 
	dp_sktr_10110: BOOL;
	localpusk_sktr_10110: BOOL;
	localstop_sktr_10110: BOOL;
	localstop_end_sktr_10110: BOOL;
	erraz_sktr_10110: BOOL;
	run_sktr_10110: BOOL;
	da_sktr_10110: BOOL:= FALSE;
	hand_sktr_10110: BOOL:= FALSE;
	
// Нория 10200
	dks_noria_10200: BOOL;
	dsl1_noria_10200: BOOL;
	dsl2_noria_10200: BOOL;
	dp_noria_10200: BOOL;
	localpusk_noria_10200: BOOL;
	localstop_but_noria_10200: BOOL;
	localstop_top_noria_10200: BOOL;
	erraz_noria_10200: BOOL;
	run_noria_10200: BOOL;
	da_noria_10200: BOOL:= FALSE;
	hand_noria_10200: BOOL:= FALSE;
	
// Система аспирации АС2 10201
	erraz_AC_10201: BOOL;
	run_AC_10201: BOOL;
	da_AC_10201: BOOL:= FALSE;
	hand_AC_10201: BOOL:= FALSE;
	
// 2-х ходовая задвижка 10210 скандия
	erraz_tflap_10210: BOOL;
	tflap_scalp_10210: BOOL;
	tflap_noria_10210: BOOL;
	run_tflap_scalp_10210: BOOL;
	run_tflap_noria_10210: BOOL;
	da_tflap_10210: BOOL:= FALSE;
	hand_tflap_scalp_10210: BOOL:= FALSE;
	hand_tflap_noria_10210: BOOL:= FALSE;
	
// Нория 10400
	dks_noria_10400: BOOL;
	dsl1_noria_10400: BOOL;
	dsl2_noria_10400: BOOL;
	dp_noria_10400: BOOL;
	localpusk_noria_10400: BOOL;
	localstop_but_noria_10400: BOOL;
	localstop_top_noria_10400: BOOL;
	erraz_noria_10400: BOOL;
	run_noria_10400: BOOL;
	da_noria_10400: BOOL:= FALSE;
	hand_noria_10400: BOOL:= FALSE;
	
// Система аспирации АС3 10401
	erraz_AC_10401: BOOL;
	run_AC_10401: BOOL;
	da_AC_10401: BOOL:= FALSE;
	hand_AC_10401: BOOL:= FALSE;
	
// Конвейер скребковый 10500
	dks_sktr_10500: BOOL;
	dp_sktr_10500: BOOL;
	localpusk_sktr_10500: BOOL;
	localstop_sktr_10500: BOOL;
	localstop_end_sktr_10500: BOOL;
	erraz_sktr_10500: BOOL;
	run_sktr_10500: BOOL;
	da_sktr_10500: BOOL:= FALSE;
	hand_sktr_10500: BOOL:= FALSE;
	
// Система аспирации АС4 10501
	erraz_AC_10501: BOOL;
	run_AC_10501: BOOL;
	da_AC_10501: BOOL:= FALSE;
	hand_AC_10501: BOOL:= FALSE;
	
// Шибер конвейера 10500 (10610)
	opened_sh_10610: BOOL;
	closed_sh_10610: BOOL;
	erraz_sh_10610: BOOL;
	run_open_sh_10610: BOOL;
	run_close_sh_10610: BOOL;
	da_sh_10610: BOOL:= FALSE;
	hand_open_sh_10610: BOOL:= FALSE;
	hand_close_sh_10610: BOOL:= FALSE;
	
// Шибер конвейера 10500 (10620)
	opened_sh_10620: BOOL;
	closed_sh_10620: BOOL;
	erraz_sh_10620: BOOL;
	run_open_sh_10620: BOOL;
	run_close_sh_10620: BOOL;
	da_sh_10620: BOOL:= FALSE;
	hand_open_sh_10620: BOOL:= FALSE;
	hand_close_sh_10620: BOOL:= FALSE;
	
// Шибер конвейера 10500 (10630)
	opened_sh_10630: BOOL;
	closed_sh_10630: BOOL;
	erraz_sh_10630: BOOL;
	run_open_sh_10630: BOOL;
	run_close_sh_10630: BOOL;
	da_sh_10630: BOOL:= FALSE;
	hand_open_sh_10630: BOOL:= FALSE;
	hand_close_sh_10630: BOOL:= FALSE;
	
// Шибер конвейера 10500 (10640)
	opened_sh_10640: BOOL;
	closed_sh_10640: BOOL;
	erraz_sh_10640: BOOL;
	run_open_sh_10640: BOOL;
	run_close_sh_10640: BOOL;
	da_sh_10640: BOOL:= FALSE;
	hand_open_sh_10640: BOOL:= FALSE;
	hand_close_sh_10640: BOOL:= FALSE;
	
// 2-х ходовая заслонка 10710 Скандия
	erraz_tflap_10710: BOOL;
	tflap_bunk_20001_10710: BOOL;
	tflap_bunk_20002_10710: BOOL;
	run_tflap_bunk_20001_10710: BOOL;
	run_tflap_bunk_20002_10710: BOOL;
	da_tflap_10710: BOOL:= FALSE;
	hand_tflap_bunk_20001_10710: BOOL:= FALSE;
	hand_tflap_bunk_20002_10710: BOOL:= FALSE;
	
// 2-х ходовая заслонка 10720 Скандия
	erraz_tflap_10720: BOOL;
	tflap_bunk_20003_10720: BOOL;
	tflap_bunk_20004_10720: BOOL;
	run_tflap_bunk_20003_10720: BOOL;
	run_tflap_bunk_20004_10720: BOOL;
	da_tflap_10720: BOOL:= FALSE;
	hand_tflap_bunk_20003_10720: BOOL:= FALSE;
	hand_tflap_bunk_20004_10720: BOOL:= FALSE;
	
// 2-х ходовая заслонка 10730 Скандия
	erraz_tflap_10730: BOOL;
	tflap_bunk_20005_10730: BOOL;
	tflap_bunk_20006_10730: BOOL;
	run_tflap_bunk_20005_10730: BOOL;
	run_tflap_bunk_20006_10730: BOOL;
	da_tflap_10730: BOOL:= FALSE;
	hand_tflap_bunk_20005_10730: BOOL:= FALSE;
	hand_tflap_bunk_20006_10730: BOOL:= FALSE;
	
// 2-х ходовая заслонка 10740 Скандия
	erraz_tflap_10740: BOOL;
	tflap_bunk_20007_10740: BOOL;
	tflap_bunk_20008_10740: BOOL;
	run_tflap_bunk_20007_10740: BOOL;
	run_tflap_bunk_20008_10740: BOOL;
	da_tflap_10740: BOOL:= FALSE;
	hand_tflap_bunk_20007_10740: BOOL:= FALSE;
	hand_tflap_bunk_20008_10740: BOOL:= FALSE;
	
// Датчики верхнего уровня бункеров 101-108
	dvy_bunk_101: BOOL;
	dvy_bunk_102: BOOL;
	dvy_bunk_103: BOOL;
	dvy_bunk_104: BOOL;
	dvy_bunk_105: BOOL;
	dvy_bunk_106: BOOL;
	dvy_bunk_107: BOOL;
	dvy_bunk_108: BOOL;
	
// Датчики нижнего уровня бункеров 20001-20008
	dny_bunk_101: BOOL;
	dny_bunk_102: BOOL;
	dny_bunk_103: BOOL;
	dny_bunk_104: BOOL;
	dny_bunk_105: BOOL;
	dny_bunk_106: BOOL;
	dny_bunk_107: BOOL;
	dny_bunk_108: BOOL;
	
// конвейер скребковый 20110
	dks_sktr_20110: BOOL;
	dp_sktr_20110: BOOL;
	localpusk_sktr_20110: BOOL;
	localstop_sktr_20110: BOOL;
	localstop_end_sktr_20110: BOOL;
	erraz_sktr_20110: BOOL;
	run_sktr_20110: BOOL;
	da_sktr_20110: BOOL:= FALSE;
	hand_sktr_20110: BOOL:= FALSE;
	
// Нория 20300
	dks_noria_20300: BOOL;
	dsl1_noria_20300: BOOL;
	dsl2_noria_20300: BOOL;
	dp_noria_20300: BOOL;
	localpusk_noria_20300: BOOL;
	localstop_but_noria_20300: BOOL;
	localstop_top_noria_20300: BOOL;
	erraz_noria_20300: BOOL;
	run_noria_20300: BOOL;
	da_noria_20300: BOOL:= FALSE;
	hand_noria_20300: BOOL:= FALSE;
	
// Система аспирации АС5 20301
	erraz_AC_20301: BOOL;
	run_AC_20301: BOOL;
	da_AC_20301: BOOL:= FALSE;
	hand_AC_20301: BOOL:= FALSE;
	
// Нория 21200
	dks_noria_21200: BOOL;
	dsl1_noria_21200: BOOL;
	dsl2_noria_21200: BOOL;
	dp_noria_21200: BOOL;
	localpusk_noria_21200: BOOL;
	localstop_but_noria_21200: BOOL;
	localstop_top_noria_21200: BOOL;
	erraz_noria_21200: BOOL;
	run_noria_21200: BOOL;
	da_noria_21200: BOOL:= FALSE;
	hand_noria_21200: BOOL:= FALSE;
	
// Конвейер шнековый 21300
	dks_shnek_21300: BOOL;
	dp_shnek_21300: BOOL;
	localstop_shnek_21300: BOOL;
	erraz_shnek_21300: BOOL;
	localpusk_shnek_21300: BOOL;
	run_shnek_21300: BOOL;
	da_shnek_21300: BOOL:= FALSE;
	hand_shnek_21300: BOOL:= FALSE;
	
// Шибер конвейера 21300 (21310)
	opened_sh_21310: BOOL;
	closed_sh_21310: BOOL;
	erraz_sh_21310: BOOL;
	run_open_sh_21310: BOOL;
	run_close_sh_21310: BOOL;
	da_sh_21310: BOOL:= FALSE;
	hand_open_sh_21310: BOOL:= FALSE;
	hand_close_sh_21310: BOOL:= FALSE;
	
// Шибер конвейера 21300 (21320)
	opened_sh_21320: BOOL;
	closed_sh_21320: BOOL;
	erraz_sh_21320: BOOL;
	run_open_sh_21320: BOOL;
	run_close_sh_21320: BOOL;
	da_sh_21320: BOOL:= FALSE;
	hand_open_sh_21320: BOOL:= FALSE;
	hand_close_sh_21320: BOOL:= FALSE;
	
// Шибер конвейера 21300 (21330)
	opened_sh_21330: BOOL;
	closed_sh_21330: BOOL;
	erraz_sh_21330: BOOL;
	run_open_sh_21330: BOOL;
	run_close_sh_21330: BOOL;
	da_sh_21330: BOOL:= FALSE;
	hand_open_sh_21330: BOOL:= FALSE;
	hand_close_sh_21330: BOOL:= FALSE;
	
// Датчики верхнего уровня бункеров 201-204
	dvy_bunk_201: BOOL;
	dvy_bunk_202: BOOL;	
	dvy_bunk_203: BOOL;	
	dvy_bunk_204: BOOL;
	
// Датчики нижнего уровня бункеров 201-204
	dny_bunk_201: BOOL;
	dny_bunk_202: BOOL;	
	dny_bunk_203: BOOL;	
	dny_bunk_204: BOOL;
	
// от дробилки
	drob_shtok_podl_high: BOOL;
	drob_shtok_podl_low: BOOL;
	drob_shtok_magn_high: BOOL;
	drob_shtok_magn_low: BOOL;
	dks_drob: BOOL;
	engine_drob_right: BOOL;
	engine_drob_left: BOOL;
	work_drob: BOOL;
	errPP_drob: BOOL;
	open_door_drob_1: BOOL;
	open_door_drob_2: BOOL;
	
	run_drob_shtok_magn_high: BOOL;
	run_drob_shtok_magn_low: BOOL;
	run_drob: BOOL;
	run_drob_right: BOOL;
	run_drob_left: BOOL;
	run_drob_shtok_podl_high: BOOL;
	
	T_1_camera_drob: WORD;
	T_2_camera_drob: WORD;
	T_1_bearing_drob: WORD;
	T_2_bearing_drob: WORD;
	
	CurrTok_drob: WORD;
	
// Питатель дробилки 30200
	errpch_pit_30200: BOOL;
	run_pit_30200: BOOL;
	run_resset_pch: BOOL;
	run_pch_30200: BOOL;
	da_pit_30200: BOOL:= FALSE;
	hand_pit_30200: BOOL:= FALSE;
	
// Электровибратор на бункере 201
	erraz_vibr_bunk_201: BOOL;
	run_vibr_bunk_201: BOOL;
	da_vibr_bunk_201: BOOL:= FALSE;
	hand_vibr_bunk_201: BOOL:= FALSE;
	
// Электровибратор на бункере 203
	erraz_vibr_bunk_203: BOOL;
	run_vibr_bunk_203: BOOL;
	da_vibr_bunk_203: BOOL:= FALSE;
	hand_vibr_bunk_203: BOOL:= FALSE;
	
// Электровибратор на бункере 205
	erraz_vibr_bunk_205: BOOL;
	run_vibr_bunk_205: BOOL;
	da_vibr_bunk_205: BOOL:= FALSE;
	hand_vibr_bunk_205: BOOL:= FALSE;
	
// Электровибратор на бункере 207
	erraz_vibr_bunk_207: BOOL;
	run_vibr_bunk_207: BOOL;
	da_vibr_bunk_207: BOOL:= FALSE;
	hand_vibr_bunk_207: BOOL:= FALSE;
	
// Электровибратор на бункере 209
	erraz_vibr_bunk_209: BOOL;
	run_vibr_bunk_209: BOOL;
	da_vibr_bunk_209: BOOL:= FALSE;
	hand_vibr_bunk_209: BOOL:= FALSE;
	
// шибер 30110
	opened_sh_30110: BOOL;
	closed_sh_30110: BOOL;
	erraz_sh_30110: BOOL;
	run_open_sh_30110: BOOL;
	run_close_sh_30110: BOOL;
	da_sh_30110: BOOL:= FALSE;
	hand_open_sh_30110: BOOL:= FALSE;
	hand_close_sh_30110: BOOL:= FALSE;
	
// Датчики уровня бункера над дробилкой
	dvy_bunk_30100: BOOL;
	dny_bunk_30100: BOOL;
	
// Датчик уровня бункерa под дробилкой 
	dvy_bunk_30200: BOOL;
	
// Вентилятор системы аспирации АС6 30310
	erraz_AC_30310: BOOL;
	run_AC_30310: BOOL;
	da_AC_30310: BOOL:= FALSE;
	hand_AC_30310: BOOL:= FALSE;
	
// Конвейер шнековый 30330
	dks_shnek_30330: BOOL;
	dp_shnek_30330: BOOL;
	localstop_shnek_30330: BOOL;
	erraz_shnek_30330: BOOL;
	localpusk_shnek_30330: BOOL;
	run_shnek_30330: BOOL;
	da_shnek_30330: BOOL:= FALSE;
	hand_shnek_30330: BOOL:= FALSE;
	
// Затвор шлюзовый 30340
	dks_shluz_30340: BOOL;
	erraz_shluz_30340: BOOL;
	run_shluz_30340: BOOL;
	da_shluz_30340: BOOL:= FALSE;
	hand_shluz_30340: BOOL:= FALSE;
	
// Конвейер скребковый 30400
	dks_sktr_30400: BOOL;
	dp_sktr_30400: BOOL;
	localpusk_sktr_30400: BOOL;
	localstop_sktr_30400: BOOL;
	localstop_end_sktr_30400: BOOL;
	erraz_sktr_30400: BOOL;
	run_sktr_30400: BOOL;
	da_sktr_30400: BOOL:= FALSE;
	hand_sktr_30400: BOOL:= FALSE;
	
// Нория 30500
	dks_noria_30500: BOOL;
	dsl1_noria_30500: BOOL;
	dsl2_noria_30500: BOOL;
	dp_noria_30500: BOOL;
	localpusk_noria_30500: BOOL;
	localstop_but_noria_30500: BOOL;
	localstop_top_noria_30500: BOOL;
	erraz_noria_30500: BOOL;
	run_noria_30500: BOOL;
	da_noria_30500: BOOL:= FALSE;
	hand_noria_30500: BOOL:= FALSE;
	
// Датчики уровня бункеров смесителя
	dvy_bunk_30610: BOOL;
	dny_bunk_30610: BOOL;
	dny_bunk_30630: BOOL;

// Датчик открытия люка на бункере БО-5	
	open_door_bunk_BO5: BOOL;
	
// Смеситель горизонтальный СГП-1000 (30600)
	open_door_smes: BOOL;
	dks_smes: BOOL;
	erraz_smes: BOOL;
	run_smes: BOOL;
	da_smes: BOOL:= FALSE;
	hand_smes: BOOL:= FALSE;
	
// от смесителя поворотный клапана, бомба люк
	klap_revers_open: BOOL;
	klap_revers_close: BOOL;
	shtok_1_left_open: BOOL;
	shtok_1_left_close: BOOL;
	shtok_2_left_open: BOOL;
	shtok_2_left_close: BOOL;
	shtok_1_right_open: BOOL;
	shtok_1_right_close: BOOL;
	shtok_2_right_open: BOOL;
	shtok_2_right_close: BOOL;
	shtok_1_zamok_close: BOOL;
	shtok_1_zamok_open: BOOL;
	shtok_2_zamok_close: BOOL;
	shtok_2_zamok_open: BOOL;
	signal_err_smes: BOOL;
	
	run_klap_revers_open: BOOL;
	run_klap_revers_close: BOOL;
	run_shtok_left_open: BOOL;
	run_shtok_left_close: BOOL;
	run_shtok_right_open: BOOL;
	run_shtok_right_close: BOOL;
	run_open_zamok: BOOL;
	run_close_zamok: BOOL;
	
// Конвейер шнековый 30640
	dks_shnek_30640: BOOL;
	dp_shnek_30640: BOOL;
	localstop_shnek30640: BOOL;
	erraz_shnek_30640: BOOL;
	localpusk_shnek_30640: BOOL;
	run_shnek_30640: BOOL;
	da_shnek_30640: BOOL:= FALSE;
	hand_shnek_30640: BOOL:= FALSE;
	
// Вентиляция аспирации АС7
	erraz_AC_7: BOOL;
	run_AC_7: BOOL;
	da_AC_7: BOOL:= FALSE;
	hand_AC_7: BOOL:= FALSE;
	
// Затвор шлюзовой аспирации АС-7_1
	dks_shluz_AC_7_1: BOOL;
	erraz_shluz_AC_7_1: BOOL;
	run_shluz_AC_7_1: BOOL;
	da_shluz_AC_7_1: BOOL:= FALSE;
	hand_shluz_AC_7_1: BOOL:= FALSE;
	
// Затвор шлюзовой аспирации АС-7_2
	dks_shluz_AC_7_2: BOOL;
	erraz_shluz_AC_7_2: BOOL;
	run_shluz_AC_7_2: BOOL;
	da_shluz_AC_7_2: BOOL:= FALSE;
	hand_shluz_AC_7_2: BOOL:= FALSE;
	
// Нория 30700
	dks_noria_30700: BOOL;
	dsl1_noria_30700: BOOL;
	dsl2_noria_30700: BOOL;
	dp_noria_30700: BOOL;
	localpusk_noria_30700: BOOL;
	localstop_but_noria_30700: BOOL;
	localstop_top_noria_30700: BOOL;
	erraz_noria_30700: BOOL;
	run_noria_30700: BOOL;
	da_noria_30700: BOOL:= FALSE;
	hand_noria_30700: BOOL:= FALSE;
	
// Система аспирации АС-8 (30701)
	erraz_AC_30701: BOOL;
	run_AC_30701: BOOL;
	da_AC_30701: BOOL:= FALSE;
	hand_AC_30701: BOOL:= FALSE;

// Конвейер скребковый 30900
	dp_sktr_30900: BOOL;
	localpusk_sktr_30900: BOOL;
	localstop_sktr_30900: BOOL;
	erraz_sktr_30900: BOOL;
	dks_sktr_30900: BOOL;
	localstop_end_sktr_30900: BOOL;
	run_sktr_30900: BOOL;
	da_sktr_30900: BOOL:= FALSE;
	hand_sktr_30900: BOOL:= FALSE;
	
// Система аспирации АС-9 (30901)
	erraz_AC_30901: BOOL;
	run_AC_30901: BOOL;
	da_AC_30901: BOOL:= FALSE;
	hand_AC_30901: BOOL:= FALSE;
	
// Шибер конвейера 30900 (30910)
	opened_sh_30910: BOOL;
	closed_sh_30910: BOOL;
	erraz_sh_30910: BOOL;
	run_open_sh_30910: BOOL;
	run_close_sh_30910: BOOL;
	da_sh_30910: BOOL:= FALSE;
	hand_open_sh_30910: BOOL:= FALSE;
	hand_close_sh_30910: BOOL:= FALSE;
	
// Шибер конвейера 30900 (30920)
	opened_sh_30920: BOOL;
	closed_sh_30920: BOOL;
	erraz_sh_30920: BOOL;
	run_open_sh_30920: BOOL;
	run_close_sh_30920: BOOL;
	da_sh_30920: BOOL:= FALSE;
	hand_open_sh_30920: BOOL:= FALSE;
	hand_close_sh_30920: BOOL:= FALSE;
	
// Шибер конвейера 30900 (30930)
	opened_sh_30930: BOOL;
	closed_sh_30930: BOOL;
	erraz_sh_30930: BOOL;
	run_open_sh_30930: BOOL;
	run_close_sh_30930: BOOL;
	da_sh_30930: BOOL:= FALSE;
	hand_open_sh_30930: BOOL:= FALSE;
	hand_close_sh_30930: BOOL:= FALSE;
	
// Шибер конвейера 30900 (30940)
	opened_sh_30940: BOOL;
	closed_sh_30940: BOOL;
	erraz_sh_30940: BOOL;
	run_open_sh_30940: BOOL;
	run_close_sh_30940: BOOL;
	da_sh_30940: BOOL:= FALSE;
	hand_open_sh_30940: BOOL:= FALSE;
	hand_close_sh_30940: BOOL:= FALSE;
	
// Конвейер скребковыйй 30800
	dks_sktr_30800: BOOL;
	dp_sktr_30800: BOOL;
	localpusk_sktr_30800: BOOL;
	localstop_sktr_30800: BOOL;
	localstop_end_sktr_30800: BOOL;
	erraz_sktr_30800: BOOL;
	run_sktr_30800: BOOL;
	da_sktr_30800: BOOL:= FALSE;
	hand_sktr_30800: BOOL:= FALSE;
	
// Шибер конвейера 30800 (30810)
	opened_sh_30810: BOOL;
	closed_sh_30810: BOOL;
	erraz_sh_30810: BOOL;
	run_open_sh_30810: BOOL;
	run_close_sh_30810: BOOL;
	da_sh_30810: BOOL:= FALSE;
	hand_open_sh_30810: BOOL:= FALSE;
	hand_close_sh_30810: BOOL:= FALSE;
	
// Шибер конвейера 30800 (30820)
	opened_sh_30820: BOOL;
	closed_sh_30820: BOOL;
	erraz_sh_30820: BOOL;
	run_open_sh_30820: BOOL;
	run_close_sh_30820: BOOL;
	da_sh_30820: BOOL:= FALSE;
	hand_open_sh_30820: BOOL:= FALSE;
	hand_close_sh_30820: BOOL:= FALSE;
	
// Конвейер бункера малых весов
	dks_shnek_21600: BOOL;
	dp_shnek_21600: BOOL;
	localstop_21600: BOOL;
	erraz_shnek_21600: BOOL;
	localpusk_shnek_21600: BOOL;
	run_shnek_21600: BOOL;
	da_shnek_21600: BOOL:= FALSE;
	hand_shnek_21600: BOOL:= FALSE;
	
// скальператор барабанный 10300
	errpch_scalp: BOOL;
	run_scalp: BOOL;
	run_resset_pch_scalp: BOOL;
	run_pch_scalp: BOOL;
	da_scalp: BOOL:= FALSE;
	hand_scalp: BOOL:= FALSE;
	
// Дазаторы 20011-20016
	errpch_doz_11_16: BOOL;
	run_pch_doz_11_16: BOOL;
	run_resset_pch_doz_11_16: BOOL;
	da_doz_pch_11_16: BOOL:= FALSE;
	
	run_doz_shnek_20011: BOOL;
	run_doz_shnek_20012: BOOL;
	run_doz_shnek_20013: BOOL;
	run_doz_shnek_20014: BOOL;
	run_doz_shnek_20015: BOOL;
	run_doz_shnek_20016: BOOL;
	
	dp_doz_shnek_20011: BOOL;
	localstop_doz_shnek_20011: BOOL;
	dp_doz_shnek_20012: BOOL;
	localstop_doz_shnek_20012: BOOL;
	dp_doz_shnek_20013: BOOL;
	localstop_doz_shnek_20013: BOOL;
	dp_doz_shnek_20014: BOOL;
	localstop_doz_shnek_20014: BOOL;
	dp_doz_shnek_20015: BOOL;
	localstop_doz_shnek_20015: BOOL;
	dp_doz_shnek_20016: BOOL;
	localstop_doz_shnek_20016: BOOL;
	
	da_doz_shnek_20011: BOOL:= FALSE;
	da_doz_shnek_20012: BOOL:= FALSE;
	da_doz_shnek_20013: BOOL:= FALSE;
	da_doz_shnek_20014: BOOL:= FALSE;
	da_doz_shnek_20015: BOOL:= FALSE;
	da_doz_shnek_20016: BOOL:= FALSE;
	da_doz_shnek_20017: BOOL:= FALSE;
	da_doz_shnek_20018: BOOL:= FALSE;
	
	hand_doz_shnek_20011: BOOL:= FALSE;
	hand_doz_shnek_20012: BOOL:= FALSE;
	hand_doz_shnek_20013: BOOL:= FALSE;
	hand_doz_shnek_20014: BOOL:= FALSE;
	hand_doz_shnek_20015: BOOL:= FALSE;
	hand_doz_shnek_20016: BOOL:= FALSE;
	hand_doz_shnek_20017: BOOL:= FALSE;
	hand_doz_shnek_20018: BOOL:= FALSE;
	
// Дазаторы 20017-20018
	errpch_doz_17_18: BOOL;
	run_pch_doz_17_18: BOOL;
	run_resset_pch_doz_17_18: BOOL;
	da_doz_pch_17_18: BOOL:= FALSE;
	
	run_doz_shnek_20017: BOOL;
	run_doz_shnek_20018: BOOL;
	
	dp_doz_shnek_20017: BOOL;
	localstop_doz_shnek_20017: BOOL;
	dp_doz_shnek_20018: BOOL;
	localstop_doz_shnek_20018: BOOL;

// Дазатор 21510-21540
	errpch_doz_shnek_51_54: BOOL;
	run_pch_doz_shnek_51_54: BOOL;
	run_resset_pch_doz_shnek_51_54: BOOL;
	da_doz_shnek_51_54: BOOL:= FALSE;
	
	run_doz_shnek_21510: BOOL;
	run_doz_shnek_21520: BOOL;
	run_doz_shnek_21530: BOOL;
	run_doz_shnek_21540: BOOL;
	
	dp_doz_shnek_21510: BOOL;
	localstop_doz_shnek_21510: BOOL;
	dp_doz_shnek_21520: BOOL;
	localstop_doz_shnek_21520: BOOL;
	dp_doz_shnek_21530: BOOL;
	localstop_doz_shnek_21530: BOOL;
	dp_doz_shnek_21540: BOOL;
	localstop_doz_shnek_21540: BOOL;
	
// Дазатор 21405-21409
	errpch_doz_shnek_5_9: BOOL;
	run_pch_doz_shnek_5_9: BOOL;
	run_resset_pch_doz_shnek_5_9: BOOL;
	da_doz_shnek_5_9: BOOL:= FALSE;
	
	run_doz_shnek_21405: BOOL;
	run_doz_shnek_21406: BOOL;
	run_doz_shnek_21407: BOOL;
	run_doz_shnek_21408: BOOL;
	run_doz_shnek_21409: BOOL;
	
	localstop_doz_shnek_21405: BOOL;
	localstop_doz_shnek_21406: BOOL;
	localstop_doz_shnek_21407: BOOL;
	localstop_doz_shnek_21408: BOOL;
	localstop_doz_shnek_21409: BOOL;
	
// Датчики верхнего уровня готовой продукции
	dvy_bunk_401: BOOL;
	dvy_bunk_402: BOOL;
	dvy_bunk_403: BOOL;
	dvy_bunk_404: BOOL;
	dvy_bunk_405: BOOL;
	dvy_bunk_406: BOOL;
	
// Датчики нижнего уровня готовой продукции
	dny_bunk_401: BOOL;
	dny_bunk_402: BOOL;
	dny_bunk_403: BOOL;
	dny_bunk_404: BOOL;
	dny_bunk_405: BOOL;
	dny_bunk_406: BOOL;
	
// Вентиляторы фильтр-шкафоф завальной ямы
	localpusk_fan_hole: BOOL;
	localstop_fan_hole: BOOL;
	erraz_AC1_1_1: BOOL;
	erraz_AC2_1_1: BOOL;
	erraz_AC3_1_1: BOOL;
	erraz_AC1_1_2: BOOL;
	erraz_AC2_1_2: BOOL;
	erraz_AC3_1_2: BOOL;
	run_fans_AC_hole: BOOL;
	da_fans_AC_hole: BOOL:= FALSE;
	hand_fans_AC_hole: BOOL:= FALSE;
	
// Конвейер 30330
	errpch_sktr_30330: BOOL;
	run_pch_sktr_30330: BOOL;
	run_resset_pch_sktr_30330: BOOL;
	da_sktr_30330: BOOL:= FALSE;
	hand_sktr_30330: BOOL:= FALSE;
	
// Датчик нижнего уровня завальной ямы
	dny_hole: BOOL;
	
// Конвейер 30640
	errpch_sktr_30640: BOOL;
	run_pch_sktr_30640: BOOL;
	run_resset_pch_sktr_30640: BOOL;
	da_sktr_30640: BOOL:= FALSE;
	hand_sktr_30640: BOOL:= FALSE;
	
// Весы большие
	W1_Big: WORD;
	W2_Big: WORD;
	Weight_Big: Real_word;
	CurrWeight_Big: REAL;	// Вес на больших весах
// Весы средние
	W1_Midle: WORD;
	W2_Midle: WORD;
	Weight_Midle: Real_word;
	CurrWeight_Midle: REAL;	// Вес на средних весах
	
END_VAR

// PLC_241/Application/ErrList
VAR_GLOBAL
// Конвейер завальной ямы 10110
	errDKS_SKTR_10110: BOOL;
	errDP_SKTR_10110: BOOL;	
	
// Нория 10200
	errDKS_noria_10200: BOOL;
	errDSL1_noria_10200: BOOL;
	errDSL2_noria_10200: BOOL;
	errDP_noria_10200: BOOL;
	
// Нория 10400
	errDKS_noria_10400: BOOL;
	errDSL1_noria_10400: BOOL;
	errDSL2_noria_10400: BOOL;
	errDP_noria_10400: BOOL;

// Нория 21200
	errDKS_noria_21200: BOOL;
	errDSL1_noria_21200: BOOL;
	errDSL2_noria_21200: BOOL;
	errDP_noria_21200: BOOL;
	
// Конвейер 10500
	errDKS_SKTR_10500: BOOL;
	errDP_SKTR_10400: BOOL;	
	
// Шибер 10610 
	errLT_sh_10610: BOOL;
	errConc_sh_10610: BOOL;
	
// Шибер 10620 
	errLT_sh_10620: BOOL;
	errConc_sh_10620: BOOL;
	
// Шибер 10630 
	errLT_sh_10630: BOOL;
	errConc_sh_10630: BOOL;
	
// Шибер 10640 
	errLT_sh_10640: BOOL;
	errConc_sh_10640: BOOL;
	
// Шибер 21310 
	errLT_sh_21310: BOOL;
	errConc_sh_21310: BOOL;
	
// Шибер 21320 
	errLT_sh_21320: BOOL;
	errConc_sh_21320: BOOL;
	
// Шибер 21330 
	errLT_sh_21330: BOOL;
	errConc_sh_21330: BOOL;
	
// 2-х ходовой клапан КП_10210
	errLT_tflap_10210: BOOL;
	errconc_tflap_10210: BOOL;
	
// 2-х ходовой клапан КП_10710
	errLT_tflap_10710: BOOL;
	errconc_tflap_10710: BOOL;
	
// 2-х ходовой клапан КП_10720
	errLT_tflap_10720: BOOL;
	errconc_tflap_10720: BOOL;
	
// 2-х ходовой клапан КП_10730
	errLT_tflap_10730: BOOL;
	errconc_tflap_10730: BOOL;
	
// 2-х ходовой клапан КП_10740
	errLT_tflap_10740: BOOL;
	errconc_tflap_10740: BOOL;
	
// Шнек 21300
	errDKS_shnek_21300: BOOL;
	errDP_shnek_21300: BOOL;
	
// Шнек Дозатор 20011
	errDP_doz_shnek_20011: BOOL;
// Шнек Дозатор 20012
	errDP_doz_shnek_20012: BOOL;
// Шнек Дозатор 20013
	errDP_doz_shnek_20013: BOOL;
// Шнек Дозатор 20014
	errDP_doz_shnek_20014: BOOL;
// Шнек Дозатор 20015
	errDP_doz_shnek_20015: BOOL;
// Шнек Дозатор 20016
	errDP_doz_shnek_20016: BOOL;
// Шнек Дозатор 20017
	errDP_doz_shnek_20017: BOOL;
// Шнек Дозатор 20018
	errDP_doz_shnek_20018: BOOL;
	
// Конвейер выгрубной од большими весами 20110
	errDKS_sktr_20110: BOOL;
	errDP_sktr_20110: BOOL;
	
END_VAR

// PLC_241/Application/Pozition_flap
VAR_GLOBAL
	// 2-х ходовая 10210
		stPoz_scalp_10210: BOOL;
		stPoz_noria_10210: BOOL;
		
	// 2-х ходовая 10710
		stPoz_bunk1_10710: BOOL;
		stPoz_bunk2_10710: BOOL;
		
	// 2-х ходовая 10720
		stPoz_bunk3_10720: BOOL;
		stPoz_bunk4_10720: BOOL;
		
	// 2-х ходовая 10730
		stPoz_bunk5_10730: BOOL;
		stPoz_bunk6_10730: BOOL;
		
	// 2-х ходовая 10740
		stPoz_bunk7_10740: BOOL;
		stPoz_bunk8_10740: BOOL;
END_VAR

// PLC_241/Application/PersistentVars
VAR_GLOBAL PERSISTENT RETAIN
END_VAR

// PLC_241/Application/BIND
PROGRAM BIND
VAR
	test: DWORD;
	TON_1: TON;
	TON_2: TON;
	TON_3: TON;
	TON_4: TON;
	TON_5: TON;
	TON_6: TON;
	TON_7: TON;
	TON_8: TON;
	TON_9: TON;
	TON_10: TON;
	TON_11: TON;
	TON_12: TON;
	TON_13: TON;
	TON_14: TON;
	TON_15: TON;
	TON_16: TON;
	TON_17: TON;
	TON_18: TON;
	TON_19: TON;
	TON_20: TON;
	TON_21: TON;
	TON_22: TON;
	TON_23: TON;
	TON_24: TON;
	TON_25: TON;
	TON_26: TON;
	TON_27: TON;
	TON_28: TON;
	TON_29: TON;
	TON_30: TON;
	TON_31: TON;
	TON_32: TON;
	TON_33: TON;
	TON_34: TON;
	TON_35: TON;
	TON_36: TON;
	TON_37: TON;
	TON_38: TON;
	TON_39: TON;
	TON_40: TON;
	TON_41: TON;
	TON_42: TON;
	TON_43: TON;
	TON_44: TON;
	TON_45: TON;
	TON_46: TON;
	TON_47: TON;
	TON_48: TON;
	TON_49: TON;
	TON_50: TON;
END_VAR

	errbtnpusk:= NOT x0_0;
	emerstop_shu:= NOT x0_1;
	emerstop_scalp:= NOT x0_2;
	emerstop_drob:= NOT x0_3;
	emerstop_smes:= NOT x0_4;
	emerstop_ubload_bunk:= NOT x0_5;
	errrkf:= NOT x0_6;
	
	y0_0:= run_sirena;
	y0_1:= run_alarm;
	
// Конвейер скребковый 
	dp_sktr_10110:= NOT x0_7;
	localpusk_sktr_10110:= x0_8;
	localstop_sktr_10110:= NOT x0_9;
	localstop_end_sktr_10110:= NOT x0_10;
	erraz_sktr_10110:= NOT x0_11;
	y0_3:= run_sktr_10110;
	
// Нория 10200
	dks_noria_10200:= x0_12;
	dsl1_noria_10200:= NOT x0_13;
	dsl2_noria_10200:= NOT x0_14;
	dp_noria_10200:= NOT x0_15;
	localpusk_noria_10200:= x0_16;
	localstop_but_noria_10200:= NOT x0_17;
	localstop_top_noria_10200:= NOT x0_18;
	erraz_noria_10200:= NOT x0_19;
	y0_4:= run_noria_10200;

// Система аспирации АС2 10201	
	erraz_AC_10201:= NOT x0_20;
	y0_5:= run_AC_10201;

// 2-х ходовая задвижка 10210 скандия	
	erraz_tflap_10210:= NOT x0_21;
	tflap_scalp_10210:= x0_22;
	tflap_noria_10210:= x0_23;
	y0_6:= run_tflap_scalp_10210;
	y0_7:= run_tflap_noria_10210;

// Нория 10400	
	dks_noria_10400:= x1_0;
	dsl1_noria_10400:= NOT x1_1;
	dsl2_noria_10400:= NOT x1_2;
	dp_noria_10400:= NOT x1_3;
	localpusk_noria_10400:= x1_4;
	localstop_but_noria_10400:= NOT x1_5;
	localstop_top_noria_10400:= NOT x1_6;
	erraz_noria_10400:= NOT x1_7;
	y0_8:= run_noria_10400;
	
// Система аспирации АС3 10401	
	erraz_AC_10401:= NOT x1_8;
	y0_9:= run_AC_10401;

// Конвейер скребковый 10500
	dks_sktr_10500:= x1_9;
	dp_sktr_10500:= NOT x1_10;
	localpusk_sktr_10500:= x1_11;
	localstop_sktr_10500:= NOT x1_12;
	localstop_end_sktr_10500:= NOT x1_13;
	erraz_sktr_10500:= NOT x1_14;
	y0_10:= run_sktr_10500;
	
// Система аспирации АС4 10501
	erraz_AC_10501:= NOT x1_15;
	y0_11:= run_AC_10501;

// Шибер конвейера 10500 (10610)
	opened_sh_10610:= NOT x1_16;
	closed_sh_10610:= NOT x1_17;
	erraz_sh_10610:= NOT x1_18;
	y0_12:= run_open_sh_10610;
	y0_13:= run_close_sh_10610;

// Шибер конвейера 10500 (10620)
	opened_sh_10620:= NOT x1_19;
	closed_sh_10620:= NOT x1_20;
	erraz_sh_10620:= NOT x1_21;
	y0_14:= run_open_sh_10620;
	y0_15:= run_close_sh_10620;
	
// Шибер конвейера 10500 (10630)
	opened_sh_10630:= NOT x1_22;
	closed_sh_10630:= NOT x1_23;
	erraz_sh_10630:= NOT x1_24;
	y6_0:= run_open_sh_10630;
	y6_1:= run_close_sh_10630;
	
// Шибер конвейера 10500 (10640)
	opened_sh_10640:= NOT x1_25;
	closed_sh_10640:= NOT x1_26;
	erraz_sh_10640:= NOT x1_27;
	y6_2:= run_open_sh_10640;
	y6_3:= run_close_sh_10640;

// 2-х ходовая заслонка 10710 Скандия
	erraz_tflap_10710:= NOT x1_28;
	tflap_bunk_20001_10710:= x1_29;
	tflap_bunk_20002_10710:= x1_30;
	y6_4:= run_tflap_bunk_20001_10710;
	y6_5:= run_tflap_bunk_20002_10710;
	
// 2-х ходовая заслонка 10720 Скандия
	erraz_tflap_10720:= NOT x1_31;
	tflap_bunk_20003_10720:= x2_0;
	tflap_bunk_20004_10720:= x2_1;
	y6_6:= run_tflap_bunk_20003_10720;
	y6_7:= run_tflap_bunk_20004_10720;
	
// 2-х ходовая заслонка 10730 Скандия
	erraz_tflap_10730:= NOT x2_2;
	tflap_bunk_20005_10730:= x2_3;
	tflap_bunk_20006_10730:= x2_4;
	y6_8:= run_tflap_bunk_20005_10730;
	y6_9:= run_tflap_bunk_20006_10730;
	
// 2-х ходовая заслонка 10740 Скандия
	erraz_tflap_10740:= NOT x2_5;
	tflap_bunk_20007_10740:= x2_6;
	tflap_bunk_20008_10740:= x2_7;
	y6_10:= run_tflap_bunk_20007_10740;
	y6_11:= run_tflap_bunk_20008_10740;
	
// Датчики верхнего уровня бункеров 101-108
	TON_1(IN:= NOT x2_8, PT:= WORD_TO_TIME(timeDVY_load*100), Q=> dvy_bunk_101);	
	TON_2(IN:= NOT x2_9, PT:= WORD_TO_TIME(timeDVY_load*100), Q=> dvy_bunk_102);
	TON_3(IN:= NOT x2_10, PT:= WORD_TO_TIME(timeDVY_load*100), Q=> dvy_bunk_103);
	TON_4(IN:= NOT x2_11, PT:= WORD_TO_TIME(timeDVY_load*100), Q=> dvy_bunk_104);
	TON_5(IN:= NOT x2_12, PT:= WORD_TO_TIME(timeDVY_load*100), Q=> dvy_bunk_105);
	TON_6(IN:= NOT x2_13, PT:= WORD_TO_TIME(timeDVY_load*100), Q=> dvy_bunk_106);
	TON_7(IN:= NOT x2_14, PT:= WORD_TO_TIME(timeDVY_load*100), Q=> dvy_bunk_107);
	TON_8(IN:= NOT x2_15, PT:= WORD_TO_TIME(timeDVY_load*100), Q=> dvy_bunk_108);
	
// Датчики нижнего уровня бункеров 20001-20008
	TON_9(IN:= NOT x2_16, PT:= WORD_TO_TIME(timeDNU_load*100), Q=> dny_bunk_101);	
	TON_10(IN:= NOT x2_17, PT:= WORD_TO_TIME(timeDNU_load*100), Q=> dny_bunk_102);
	TON_11(IN:= NOT x2_18, PT:= WORD_TO_TIME(timeDNU_load*100), Q=> dny_bunk_103);
	TON_12(IN:= NOT x2_19, PT:= WORD_TO_TIME(timeDNU_load*100), Q=> dny_bunk_104);
	TON_13(IN:= NOT x2_20, PT:= WORD_TO_TIME(timeDNU_load*100), Q=> dny_bunk_105);
	TON_14(IN:= NOT x2_21, PT:= WORD_TO_TIME(timeDNU_load*100), Q=> dny_bunk_106);
	TON_15(IN:= NOT x2_22, PT:= WORD_TO_TIME(timeDNU_load*100), Q=> dny_bunk_107);
	TON_16(IN:= NOT x2_23, PT:= WORD_TO_TIME(timeDNU_load*100), Q=> dny_bunk_108);
	
// конвейер скребковый 20110
	dks_sktr_20110:= x2_24;
	dp_sktr_20110:= NOT x2_25;
	localpusk_sktr_20110:= x2_26;
	localstop_sktr_20110:= NOT x2_27;
	localstop_end_sktr_20110:= x2_28;
	erraz_sktr_20110:= NOT x2_29;
	y6_12:= run_sktr_20110;
	
// Нория 20300
	dks_noria_20300:= x2_30;
	dsl1_noria_20300:= NOT x2_31;
	dsl2_noria_20300:= NOT x3_0;
	dp_noria_20300:= NOT x3_1;
	localpusk_noria_20300:= x3_2;
	localstop_but_noria_20300:= NOT x3_3;
	localstop_top_noria_20300:= NOT x3_4;
	erraz_noria_20300:= NOT x3_5;
	y6_13:= run_noria_20300;
	
// Система аспирации АС5 20301
	erraz_AC_20301:= NOT x3_6;
	y6_14:= run_AC_20301;
	
// Нория 21200
	dks_noria_21200:= x3_7;
	dsl1_noria_21200:= NOT x3_8;
	dsl2_noria_21200:= NOT x3_9;
	dp_noria_21200:= NOT x3_10;
	localpusk_noria_21200:= x3_11;
	localstop_but_noria_21200:= NOT x3_12;
	localstop_top_noria_21200:= NOT x3_13;
	erraz_noria_21200:= NOT x3_14;
	y6_15:= run_noria_21200;

// Конвейер шнековый 21300
	dks_shnek_21300:= x3_15;
	dp_shnek_21300:= NOT x3_16;
	localstop_shnek_21300:= NOT x3_17;
	erraz_shnek_21300:= NOT x3_18;
	localpusk_shnek_21300:= x3_19;
	y6_16:= run_shnek_21300;
	
// Шибер конвейера 21300 (21310)
	opened_sh_21310:= NOT x3_20;
	closed_sh_21310:= NOT x3_21;
	erraz_sh_21310:= NOT x3_22;
	y6_17:= run_open_sh_21310;
	y6_18:= run_close_sh_21310;
	
// Шибер конвейера 21300 (21320)	
	opened_sh_21320:= NOT x3_23;
	closed_sh_21320:= NOT x3_24;
	erraz_sh_21320:= NOT x3_25;
	y6_19:= run_open_sh_21320;
	y6_20:= run_close_sh_21320;
	
// Шибер конвейера 21300 (21330)
	opened_sh_21330:= NOT x3_26;
	closed_sh_21330:= NOT x3_27;
	erraz_sh_21330:= NOT x3_28;
	y6_21:= run_open_sh_21330;
	y6_22:= run_close_sh_21330;
	
// Датчики верхнего уровня бункеров 201-204
	TON_17(IN:= NOT x3_29, PT:= WORD_TO_TIME(timeDVY_load*100), Q=> dvy_bunk_201);
	TON_18(IN:= NOT x3_30, PT:= WORD_TO_TIME(timeDVY_load*100), Q=> dvy_bunk_202);
	TON_19(IN:= NOT x4_0, PT:= WORD_TO_TIME(timeDVY_load*100), Q=> dvy_bunk_203);
	TON_20(IN:= NOT x4_1, PT:= WORD_TO_TIME(timeDVY_load*100), Q=> dvy_bunk_204);
	
// Датчики нижнего уровня бункеров 201-204
	TON_21(IN:= NOT x4_2, PT:= WORD_TO_TIME(timeDNU_load*100), Q=> dny_bunk_201);
	TON_22(IN:= NOT x4_3, PT:= WORD_TO_TIME(timeDNU_load*100), Q=> dny_bunk_202);
	TON_23(IN:= NOT x4_4, PT:= WORD_TO_TIME(timeDNU_load*100), Q=> dny_bunk_203);
	TON_24(IN:= NOT x4_5, PT:= WORD_TO_TIME(timeDNU_load*100), Q=> dny_bunk_204);
	
// от дробилки
	drob_shtok_podl_high:= x4_6;
	drob_shtok_podl_low:= x4_7;
	drob_shtok_magn_high:= x4_8;
	drob_shtok_magn_low:= x4_9;
	dks_drob:= x4_10;
	engine_drob_right:= x4_11;
	engine_drob_left:= x4_12;
	work_drob:= x4_13;
	errPP_drob:= x4_14;
	open_door_drob_1:= NOT x4_15;
	open_door_drob_2:= NOT x4_16;
	
	y6_23:= run_drob_shtok_magn_high;
	y6_24:= run_drob_shtok_magn_low;
	y6_25:= run_drob;
	y6_26:= run_drob_right;
	y6_27:= run_drob_left;
	y6_28:= run_drob_shtok_podl_high;
	
	T_1_camera_drob:= IW1_0;
	T_2_camera_drob:= IW1_1;
	T_1_bearing_drob:= IW1_2;
	T_2_bearing_drob:= IW1_3;
	
	CurrTok_drob:= IW2_0;
	
// Питатель дробилки 30200
	errpch_pit_30200:= x4_17;
	y6_29:= run_pit_30200;
	y6_30:= run_resset_pch;
	y6_31:= run_pch_30200;
	
// Электровибратор на бункере 201
	erraz_vibr_bunk_201:= NOT x4_18;
	y7_0:= run_vibr_bunk_201;
	
// Электровибратор на бункере 203
	erraz_vibr_bunk_203:= NOT x4_19;
	y7_1:= run_vibr_bunk_203;
	
// Электровибратор на бункере 205
	erraz_vibr_bunk_205:= NOT x4_20;
	y7_2:= run_vibr_bunk_205;
	
// Электровибратор на бункере 207
	erraz_vibr_bunk_207:= NOT x4_21;
	y7_3:= run_vibr_bunk_207;
	
// Электровибратор на бункере 209
	erraz_vibr_bunk_209:= NOT x4_22;
	y7_4:= run_vibr_bunk_209;
	
// шибер 30110
	opened_sh_30110:= NOT x4_23;
	closed_sh_30110:= NOT x4_24;
	erraz_sh_30110:= NOT x4_25;
	y7_5:= run_open_sh_30110;
	y7_6:= run_close_sh_30110;
	
// Датчики уровня бункера над дробилкой
	TON_25(IN:= NOT x4_26, PT:= WORD_TO_TIME(timeDVY_load*100), Q=> dvy_bunk_30100);
	TON_26(IN:= NOT x4_27, PT:= WORD_TO_TIME(timeDNU_load*100), Q=> dny_bunk_30100);
	
// Датчик уровня бункерa под дробилкой 
	TON_27(IN:= NOT x4_28, PT:= WORD_TO_TIME(timeDVY_load*100), Q=> dvy_bunk_30200);
	
// Вентилятор системы аспирации АС6 30310
	erraz_AC_30310:= NOT x4_29;
	y7_7:= run_AC_30310;
	
